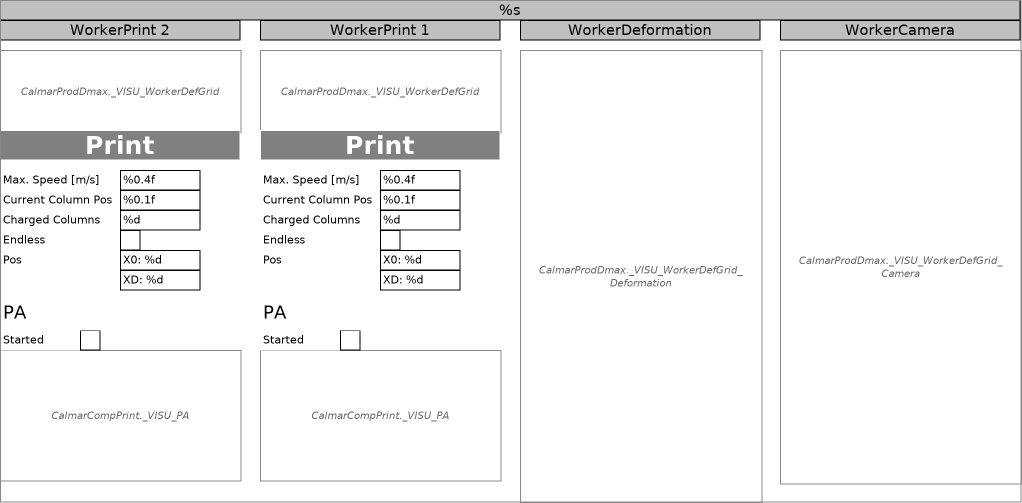
VISUALIZATION _VISU_Pm_Worker  // 1022x503
VAR_IN_OUT
	mInst : FB_PrintModule_WEU;
END_VAR
    Frame (0,50 242x404)
        shows _VISU_WorkerPrint_WEU(m_Inst := mInst.fbWorkerPrint[2])
    Frame (260,50 242x406)
        shows _VISU_WorkerPrint_WEU(m_Inst := mInst.fbWorkerPrint[1])
    Rectangle (0,20 240x20), "WorkerPrint 2"
    Rectangle (260,20 240x20), "WorkerPrint 1"
    Frame (780,50 242x434)
        shows CalmarProdDmax._VISU_WorkerDefGrid_Camera(m_Inst := mInst.fbWorkerCamera)
    Rectangle (780,20 240x20), "WorkerCamera"
    Rectangle (0,0 1020x20), "%s", text variable: mInst._pAdsPm^.aO_Name
    Rectangle (520,20 240x20), "WorkerDeformation"
    Frame (520,50 242x453)
        shows CalmarProdDmax._VISU_WorkerDefGrid_Deformation(m_Inst := mInst.fbWorkerDeformation)
END_VISUALIZATION

// ---- POUs/Projects/Machine/_VISU_MachineComm.TcVIS
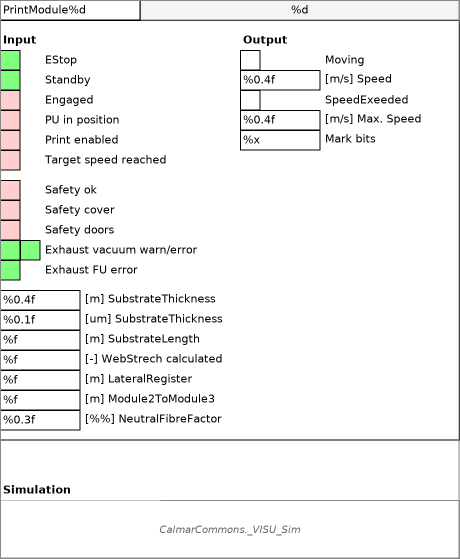
VISUALIZATION _VISU_MachineComm  // 460x559
VAR_IN_OUT
	mInst : FB_MachineComm;
END_VAR
    Rectangle (0,20 460x420)
    Frame (0,50 260x364)
        shows _VISU_MachineIn(ref := mInst.sModuleMachineState[mInst.nSelPm])
    Frame (240,50 214x110)
        shows _VISU_MachineOut(ref := mInst.sModuleMachineFeedback[mInst.nSelPm])
    Frame (0,500 460x59)
        shows CalmarCommons._VISU_Sim(mInst := mInst)
    Rectangle (240,30 160x20), "Output"
    Rectangle (0,30 160x20), "Input"
    Rectangle (0,480 160x20), "Simulation"
    Scrollbar (140,0 320x20), "%d", text variable: mInst.nSelPm
        p2245068023: iCPr_NB_PM
        p1057716461: mInst.nSelPm
    Rectangle (0,0 140x20), "PrintModule%d", text variable: PRG_PRINT.fbModuleMaster.nViewPmSel
END_VISUALIZATION

// ---- POUs/Projects/Machine/_VISU_MachineIn.TcVIS
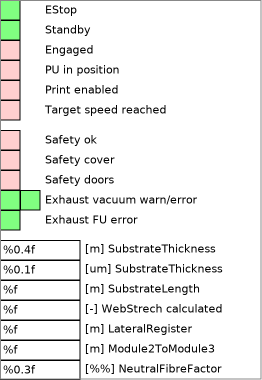
VISUALIZATION _VISU_MachineIn  // 262x380
VAR_IN_OUT
	ref : ST_ModuleMachineInterface_IN;
END_VAR
    Rectangle (0,320 80x20), "%f", text variable: ref.fLateralRegister
    Rectangle (82,320 180x18), "[m] LateralRegister"
    Rectangle (0,240 80x20), "%0.4f", text variable: ref.fSubstrateThickness
    Rectangle (82,240 180x18), "[m] SubstrateThickness"
    Rectangle (0,280 80x20), "%f", text variable: ref.fSubstrateLen
    Rectangle (82,280 180x18), "[m] SubstrateLength"
    Rectangle (0,300 80x20), "%f", text variable: ref.fWebStretchCalculated
    Rectangle (82,300 180x18), "[-] WebStrech calculated"
    Rectangle (0,340 80x20), "%f", text variable: ref.fModule2ToModule3
    Rectangle (82,340 180x18), "[m] Module2ToModule3"
    Rectangle (0,360 80x20), "%0.3f", text variable: ref.fNeutralFibreFactor
    Rectangle (82,360 180x18), "[%%] NeutralFibreFactor"
    Rectangle (42,20 180x20), "Standby"
    RoundedRectangle (0,0 20x20), colour toggle: ref.bEStop
    Rectangle (42,0 180x20), "EStop"
    RoundedRectangle (0,20 20x20), colour toggle: ref.bSleep
    RoundedRectangle (0,150 20x20), colour toggle: ref.bSafetyCoverOk
    Rectangle (42,150 180x20), "Safety cover"
    RoundedRectangle (0,170 20x20), colour toggle: ref.bServiceDoorsOk
    Rectangle (42,170 180x20), "Safety doors"
    RoundedRectangle (0,190 20x20), colour toggle: ref.bExhaustVacuumWarning
    Rectangle (42,190 180x20), "Exhaust vacuum warn/error"
    Rectangle (42,210 180x20), "Exhaust FU error"
    Rectangle (42,130 180x20), "Safety ok"
    RoundedRectangle (0,130 20x20), colour toggle: ref.bSafetyOk
    RoundedRectangle (20,190 20x20), colour toggle: ref.bExhaustVacuumError
    RoundedRectangle (0,210 20x20), colour toggle: ref.bExhaustFUError
    Rectangle (42,60 180x20), "PU in position"
    RoundedRectangle (0,60 20x20), colour toggle: ref.bUnitInPrintPosition
    Rectangle (42,40 180x20), "Engaged"
    RoundedRectangle (0,40 20x20), colour toggle: ref.bEngaged
    Rectangle (42,80 180x20), "Print enabled"
    RoundedRectangle (0,80 20x20), colour toggle: ref.bPrintEnabled
    Rectangle (42,100 180x20), "Target speed reached"
    RoundedRectangle (0,100 20x20), colour toggle: ref.bTargetSpeedReached
    Rectangle (0,260 80x20), "%0.1f", text variable: ref.fSubstrateThickness * 1_000_000
    Rectangle (82,260 180x18), "[um] SubstrateThickness"
END_VISUALIZATION

// ---- POUs/Projects/Machine/_VISU_MachineOut.TcVIS
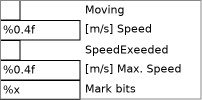
VISUALIZATION _VISU_MachineOut  // 202x100
VAR_IN_OUT
	ref : ST_ModuleMachineInterface_OUT;
END_VAR
    Rectangle (0,20 80x20), "%0.4f", text variable: ref.fSpeed
    Rectangle (82,20 120x18), "[m/s] Speed"
    Rectangle (0,60 80x20), "%0.4f", text variable: ref.fMaxSpeed
    Rectangle (82,60 120x18), "[m/s] Max. Speed"
    Rectangle (82,0 120x20), "Moving"
    RoundedRectangle (0,40 20x20), colour toggle: ref.bSpeedExeeded
    Rectangle (82,40 120x20), "SpeedExeeded"
    RoundedRectangle (0,0 20x20), colour toggle: ref.bMoving
    Rectangle (0,80 80x20), "%x", text variable: ref.nPrintMarkPosBits
    Rectangle (82,80 120x18), "Mark bits"
END_VISUALIZATION

// ---- POUs/Projects/Print/_Test/_VISU_PrgPrint_test.TcVIS
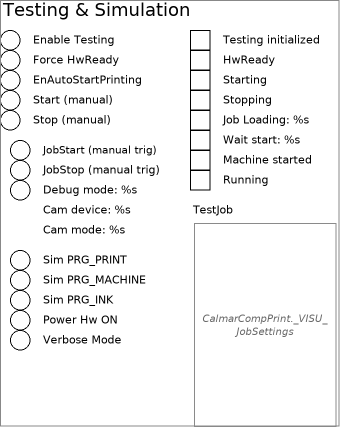
VISUALIZATION _VISU_PrgPrint_test  // 340x427
VAR_IN_OUT
	mInst : FB_PrgPrint_test;
END_VAR
    Ellipse (0,30 20x20)
        toggle mInst._bEnTesting
    Rectangle (30,30 120x20), "Enable Testing"
    Ellipse (0,70 20x20)
        toggle mInst._bEnAutoStartPrinting
    Rectangle (30,70 120x20), "EnAutoStartPrinting"
    Ellipse (10,180 20x20)
        toggle mInst._bEnVerboseMode
    Rectangle (40,180 120x20), "Debug mode: %s", text variable: mInst._eLogLevel
    Ellipse (10,270 20x20)
        toggle mInst._bSimPrgMachine
    Rectangle (40,270 120x20), "Sim PRG_MACHINE"
    Ellipse (10,290 20x20)
        toggle mInst._bSimPrgInk
    Rectangle (40,290 120x20), "Sim PRG_INK"
    Ellipse (10,250 20x20)
        toggle mInst._bSimPrgPrint
    Rectangle (40,250 120x20), "Sim PRG_PRINT"
    RoundedRectangle (190,30 20x20), colour toggle: mInst.bInitialized
    Rectangle (220,30 120x20), "Testing initialized"
    RoundedRectangle (190,50 20x20), tooltip "All enabled CBs are in OP", colour toggle: mInst.bHwReady
    Rectangle (220,50 120x20), "HwReady"
    RoundedRectangle (190,70 20x20), colour toggle: mInst.bStarting
    Rectangle (220,70 120x20), "Starting"
    RoundedRectangle (190,90 20x20), colour toggle: mInst.bStopping
    Rectangle (220,90 120x20), "Stopping"
    RoundedRectangle (190,170 20x20), colour toggle: mInst.bRunning
    Rectangle (220,170 120x20), "Running"
    Rectangle (220,110 120x20), "Job Loading: %s", tooltip "Timeout after: %s", text variable: mInst.LoadTestJob.tExecute.ET
        p4168582468: mInst.LoadTestJob.tExecute.PT
    RoundedRectangle (190,110 20x20), colour toggle: mInst.LoadTestJob.bbusy
    Rectangle (220,130 120x20), "Wait start: %s", text variable: mInst.TestStartSequence.tWaitJobStart.ET
    RoundedRectangle (190,130 20x20), colour toggle: mInst.TestStartSequence.tWaitJobStart.IN
    Rectangle (40,200 120x20), "Cam device: %s", text variable: mInst.eCameraDevice
        OnMouseClick: write the text variable via Default
    Rectangle (40,220 120x20), "Cam mode: %s", text variable: mInst.eCameraMode
        OnMouseClick: write the text variable via Default
    Ellipse (0,90 20x20)
        toggle mInst.bStart
    Rectangle (30,90 120x20), "Start (manual)"
    Ellipse (0,110 20x20)
        toggle mInst.bStop
    Rectangle (30,110 120x20), "Stop (manual)"
    Rectangle (0,0 200x20), "Testing & Simulation"
    Ellipse (10,140 20x20)
        tap mInst._pAdsPu^.sI_Start.bI_Command
        toggle mInst.bStart
    Rectangle (40,140 120x20), "JobStart (manual trig)"
    Ellipse (10,160 20x20)
        tap mInst._pAdsPu^.sI_Stop.bI_Command
        toggle mInst.bStop
    Rectangle (40,160 120x20), "JobStop (manual trig)"
    Frame (194,223 142x204)
        shows CalmarCompPrint._VISU_JobSettings(mInst := mInst.sJobConfig)
    RoundedRectangle (190,150 20x20), colour toggle: mInst.bRunMachine
    Rectangle (220,150 120x20), "Machine started"
    Rectangle (190,200 120x20), "TestJob"
    Ellipse (0,50 20x20)
        toggle mInst._bForceHwReady
    Rectangle (30,50 120x20), "Force HwReady"
    Ellipse (10,310 20x20)
        toggle mInst.bO_Power24V_ON
    Rectangle (40,310 120x20), "Power Hw ON"
    Ellipse (10,330 20x20)
        toggle mInst._bEnVerboseMode
    Rectangle (40,330 120x20), "Verbose Mode"
END_VISUALIZATION

// ---- VISUs/Projects/InkSystem/VISU_ADS_INKSTORAGE_TANK_DVT.TcVIS
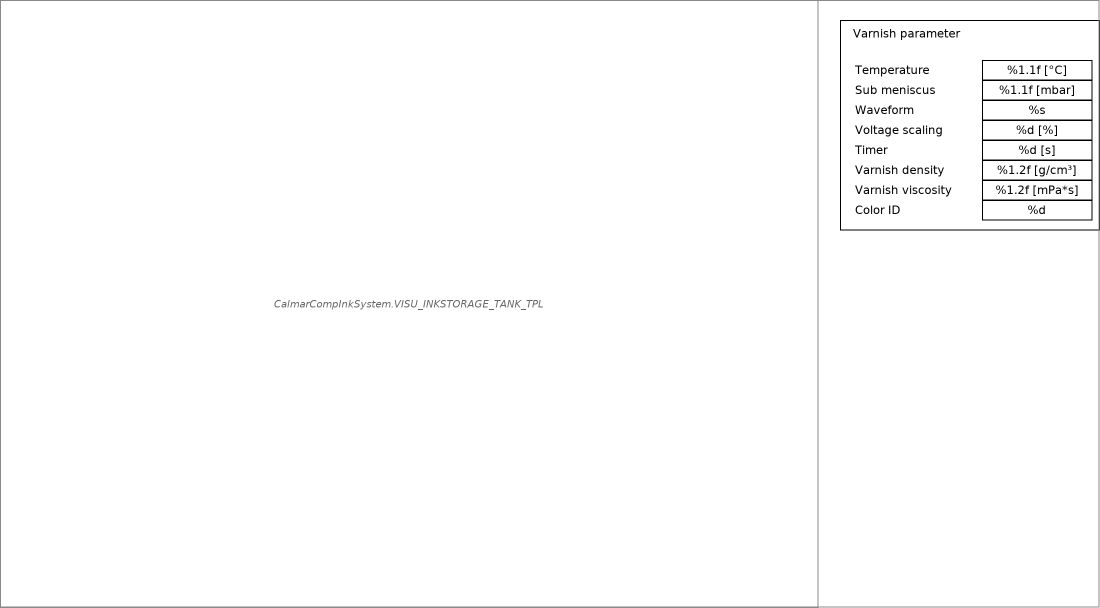
VISUALIZATION VISU_ADS_INKSTORAGE_TANK_DVT  // 1100x608
    Frame (0,0 818x608)
        shows CalmarCompInkSystem.VISU_INKSTORAGE_TANK_TPL(m_Idx_Max := CONFIGURATION.iCIk_NB_INKSTORAGE_TANK, m_ModId_StAdsStorageTank := PRG_INK.sAdsIkInkStorageTank[PRG_INK.iL_Sel_InkStorTank], m_Idx := PRG_INK.iL_Sel_InkStorTank, m_EnableBalanceLink := PRG_INK.bI_EnableBalanceLink, m_RefreshRate := PRG_INK.iI_RefreshRate, m_BalanceOffset := PRG_INK.fL_BalanceOffset[PRG_INK.iL_Sel_InkStorTank], m_CorrectionValue := PRG_INK.fI_CorrectionValue, m_MixerFeedbackExist := PRG_INK.bL_MixerFeedbackExist, m_MixerPulseIndicator := PRG_INK.bL_MixerPulseIndicator[PRG_INK.iL_Sel_InkStorTank], m_AckMixerPulseError := PRG_INK.bL_AckMixerPulseError[PRG_INK.iL_Sel_InkStorTank], m_MixerOnTime := PRG_INK.fL_MixerOnTime, m_MixerWaitTime := PRG_INK.fL_MixerWaitTime)
    Rectangle (840,20 260x210)
    Rectangle (982,60 110x20), "%1.1f [°C]", text variable: PRG_INK.sAdsIkInkStorageTank[PRG_INK.iL_Sel_InkStorTank].sI_InkParameter.sTemperature.fI_Val
        OnMouseDown: write the text variable via Edit, min PRG_INK.sAdsIkInkStorageTank[PRG_INK.iL_Sel_InkStorTank].sI_MaintenanceTimeout.lC_Min, max PRG_INK.sAdsIkInkStorageTank[PRG_INK.iL_Sel_InkStorTank].sI_MaintenanceTimeout.lC_Max
    Rectangle (852,60 130x20), "Temperature"
    Rectangle (850,25 191x17), "Varnish parameter"
    Rectangle (982,80 110x20), "%1.1f [mbar]", text variable: PRG_INK.sAdsIkInkStorageTank[PRG_INK.iL_Sel_InkStorTank].sI_InkParameter.sMeniscus.fI_Val
        OnMouseDown: write the text variable via Edit, min PRG_INK.sAdsIkInkStorageTank[PRG_INK.iL_Sel_InkStorTank].sI_InkParameter.sMeniscus.fC_Min, max PRG_INK.sAdsIkInkStorageTank[PRG_INK.iL_Sel_InkStorTank].sI_InkParameter.sMeniscus.fC_Max
    Rectangle (852,80 130x20), "Sub meniscus"
    Rectangle (982,100 110x20), "%s", text variable: PRG_INK.sAdsIkInkStorageTank[PRG_INK.iL_Sel_InkStorTank].sI_InkParameter.aWaveform
        OnMouseDown: write the text variable via Edit, min PRG_INK.sAdsIkInkStorageTank[PRG_INK.iL_Sel_InkStorTank].sI_MaintenanceTimeout.lC_Min, max PRG_INK.sAdsIkInkStorageTank[PRG_INK.iL_Sel_InkStorTank].sI_MaintenanceTimeout.lC_Max
    Rectangle (852,100 130x20), "Waveform"
    Rectangle (982,120 110x20), "%d [%]", text variable: PRG_INK.sAdsIkInkStorageTank[PRG_INK.iL_Sel_InkStorTank].sI_InkParameter.iVoltage
        OnMouseDown: write the text variable via Edit, min PRG_INK.sAdsIkInkStorageTank[PRG_INK.iL_Sel_InkStorTank].sI_MaintenanceTimeout.lC_Min, max PRG_INK.sAdsIkInkStorageTank[PRG_INK.iL_Sel_InkStorTank].sI_MaintenanceTimeout.lC_Max
    Rectangle (852,120 130x20), "Voltage scaling"
    Rectangle (982,140 110x20), "%d [s]", text variable: PRG_INK.sAdsIkInkStorageTank[PRG_INK.iL_Sel_InkStorTank].sI_InkParameter.iTimer
        OnMouseDown: write the text variable via Edit, min PRG_INK.sAdsIkInkStorageTank[PRG_INK.iL_Sel_InkStorTank].sI_MaintenanceTimeout.lC_Min, max PRG_INK.sAdsIkInkStorageTank[PRG_INK.iL_Sel_InkStorTank].sI_MaintenanceTimeout.lC_Max
    Rectangle (852,140 130x20), "Timer"
    Rectangle (982,160 110x20), "%1.2f [g/cm³]", text variable: PRG_INK.sAdsIkInkStorageTank[PRG_INK.iL_Sel_InkStorTank].sI_InkParameter.sDensity.fI_Val
        OnMouseDown: write the text variable via Edit, min PRG_INK.sAdsIkInkStorageTank[PRG_INK.iL_Sel_InkStorTank].sI_MaintenanceTimeout.lC_Min, max PRG_INK.sAdsIkInkStorageTank[PRG_INK.iL_Sel_InkStorTank].sI_MaintenanceTimeout.lC_Max
    Rectangle (852,160 130x20), "Varnish density"
    Rectangle (982,180 110x20), "%1.2f [mPa*s]", text variable: PRG_INK.sAdsIkInkStorageTank[PRG_INK.iL_Sel_InkStorTank].sI_InkParameter.sViscosity.fI_Val
        OnMouseDown: write the text variable via Edit, min PRG_INK.sAdsIkInkStorageTank[PRG_INK.iL_Sel_InkStorTank].sI_MaintenanceTimeout.lC_Min, max PRG_INK.sAdsIkInkStorageTank[PRG_INK.iL_Sel_InkStorTank].sI_MaintenanceTimeout.lC_Max
    Rectangle (852,180 130x20), "Varnish viscosity"
    Rectangle (982,200 110x20), "%d", text variable: PRG_INK.sAdsIkInkStorageTank[PRG_INK.iL_Sel_InkStorTank].sI_InkParameter.iColorId
        OnMouseDown: write the text variable via Edit, min PRG_INK.sAdsIkInkStorageTank[PRG_INK.iL_Sel_InkStorTank].sI_MaintenanceTimeout.lC_Min, max PRG_INK.sAdsIkInkStorageTank[PRG_INK.iL_Sel_InkStorTank].sI_MaintenanceTimeout.lC_Max
    Rectangle (852,200 130x20), "Color ID"
END_VISUALIZATION

// ---- VISUs/Projects/InkSystem/VISU_BALANCE.TcVIS
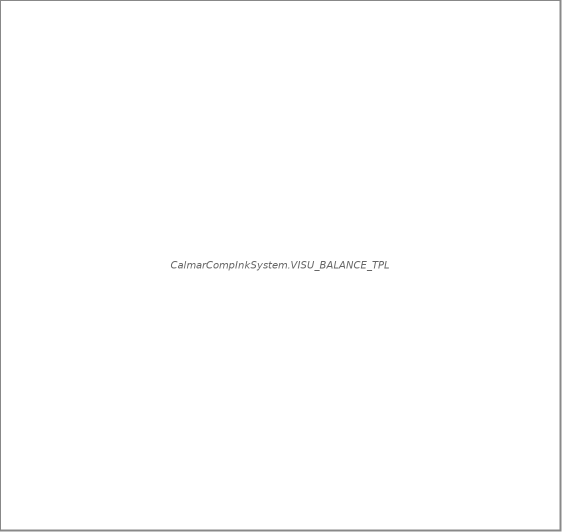
VISUALIZATION VISU_BALANCE  // 562x532
    Frame (0,0 560x530)
        shows CalmarCompInkSystem.VISU_BALANCE_TPL(m_Idx_Max := CONFIGURATION.iCIk_NB_INKBALANCE, m_ModId_StAdsStorageTank := PRG_INK.sAdsIkInkStorageTank[PRG_INK.iL_SelectedBalance], m_ModId_FbBalanceMonitor := PRG_INK.FB_Balance[PRG_INK.iL_SelectedBalance], m_Idx := PRG_INK.iL_SelectedBalance)
END_VISUALIZATION

// ---- VISUs/Projects/InkSystem/VISU_BARCODE.TcVIS
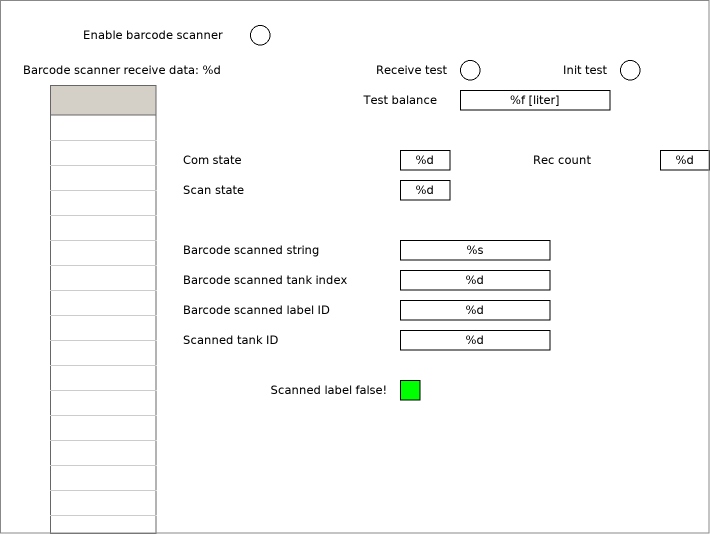
VISUALIZATION VISU_BARCODE  // 710x534
    Table (50,85 106x449), data array: PRG_INK.cI_Barcode_RxBuff
        p2232123230: PRG_INK.cI_Barcode_RxBuff[INDEX]
        p511219082: PRG_PRINT.sL_SensorResults[INDEX].yMark
        p1755163831: PRG_PRINT.sL_SensorResults[INDEX].phiMark
        p4092479075: PRG_PRINT.sL_SensorResults[INDEX].xCam
        p2237128397: PRG_PRINT.sL_SensorResults[INDEX].yCam
        p505689113: PRG_PRINT.sL_SensorResults[INDEX].phiCam
        p1757482276: PRG_PRINT.sL_SensorResults[INDEX].dx
        p4088588272: PRG_PRINT.sL_SensorResults[INDEX].dy
        p2243050616: PRG_PRINT.sL_SensorResults[INDEX].dphi
    Rectangle (20,60 240x20), "Barcode scanner receive data: %d", text variable: PRG_INK.iI_Barcode_RecDataLength
    Rectangle (400,240 150x20), "%s", text variable: PRG_INK.fb_BarcodeStoragetank.aL_ReceivedData
    Rectangle (180,240 200x20), "Barcode scanned string"
    Rectangle (400,270 150x20), "%d", text variable: PRG_INK.fb_BarcodeStoragetank.iL_ScannedStorageIndex
    Rectangle (180,270 200x20), "Barcode scanned tank index"
    Rectangle (400,300 150x20), "%d", text variable: PRG_INK.fb_BarcodeStoragetank.lL_ScannedLabel
    Rectangle (180,300 200x20), "Barcode scanned label ID"
    Rectangle (400,330 150x20), "%d", text variable: PRG_INK.sAdsIkInkStorageTank[PRG_INK.fb_BarcodeStoragetank.iL_ScannedStorageIndex].sI_InkParameter.iScannerId
        OnMouseClick: write the text variable via Default
    Rectangle (180,330 200x20), "Scanned tank ID"
    Rectangle (219,380 171x20), "Scanned label false!"
    RoundedRectangle (400,380 20x20), colour toggle: PRG_INK.fb_BarcodeStoragetank.bO_LabelScanFalse[PRG_INK.fb_BarcodeStoragetank.iL_ScannedStorageIndex]
    Rectangle (80,25 160x20), "Enable barcode scanner"
    Ellipse (250,25 20x20), colour toggle: PRG_INK.bI_EnableBarcodeScanner
        toggle PRG_INK.bI_EnableBarcodeScanner
    Rectangle (355,60 95x20), "Receive test"
    Ellipse (460,60 20x20), colour toggle: PRG_INK.bI_Barcode_DataRec
        tap PRG_INK.bI_Barcode_DataRec
    Rectangle (400,180 50x20), "%d", text variable: PRG_INK.fb_BarcodeStoragetank.iL_ScanState
        OnMouseClick: write the text variable via Default
    Rectangle (180,180 200x20), "Scan state"
    Rectangle (515,60 95x20), "Init test"
    Ellipse (620,60 20x20), colour toggle: PRG_INK.bI_Barcode_AckInit
        tap PRG_INK.bI_Barcode_AckInit
    Rectangle (400,150 50x20), "%d", text variable: PRG_INK.fb_BarcodeStoragetank.iL_COMstate
        OnMouseClick: write the text variable via Default
    Rectangle (180,150 200x20), "Com state"
    Rectangle (460,90 150x20), "%f [liter]", text variable: PRG_INK.FB_BalanceLink.fO_Readings[PRG_INK.fb_BarcodeStoragetank.iL_ScannedStorageIndex]
        OnMouseClick: write the text variable via Default
    Rectangle (329,90 111x20), "Test balance"
    Rectangle (660,150 50x20), "%d", text variable: PRG_INK.fb_BarcodeStoragetank.iL_ReceiveCount
    Rectangle (530,150 102x20), "Rec count"
END_VISUALIZATION

// ---- VISUs/Projects/InkSystem/VISU_COMM_BALANCE.TcVIS
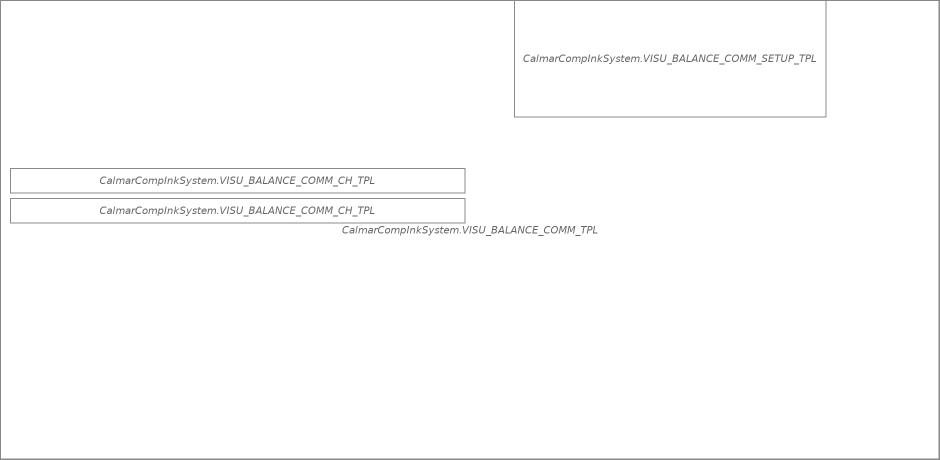
VISUALIZATION VISU_COMM_BALANCE  // 940x460
    Frame (0,0 940x460)
        shows CalmarCompInkSystem.VISU_BALANCE_COMM_TPL(m_ModId_FbBalanceComm := PRG_INK.FB_BalanceLink)
    Frame (514,0 312x117)
        shows CalmarCompInkSystem.VISU_BALANCE_COMM_SETUP_TPL(m_ModId_FbBalanceComm := PRG_INK.FB_BalanceLink)
    Frame (10,168 455x25)
        shows CalmarCompInkSystem.VISU_BALANCE_COMM_CH_TPL(m_Idx := 1, m_ModId_StAdsStorageTank := PRG_INK.sAdsIkInkStorageTank[1], m_ModId_StInkDefinition := PRG_INK.sL_InkTable[1], m_ModId_FbBalanceComm := PRG_INK.FB_BalanceLink)
    Frame (10,198 455x25)
        shows CalmarCompInkSystem.VISU_BALANCE_COMM_CH_TPL(m_Idx := 2, m_ModId_StAdsStorageTank := PRG_INK.sAdsIkInkStorageTank[2], m_ModId_StInkDefinition := PRG_INK.sL_InkTable[2], m_ModId_FbBalanceComm := PRG_INK.FB_BalanceLink)
END_VISUALIZATION

// ---- VISUs/Projects/InkSystem/VISU_HEADERTANK.TcVIS
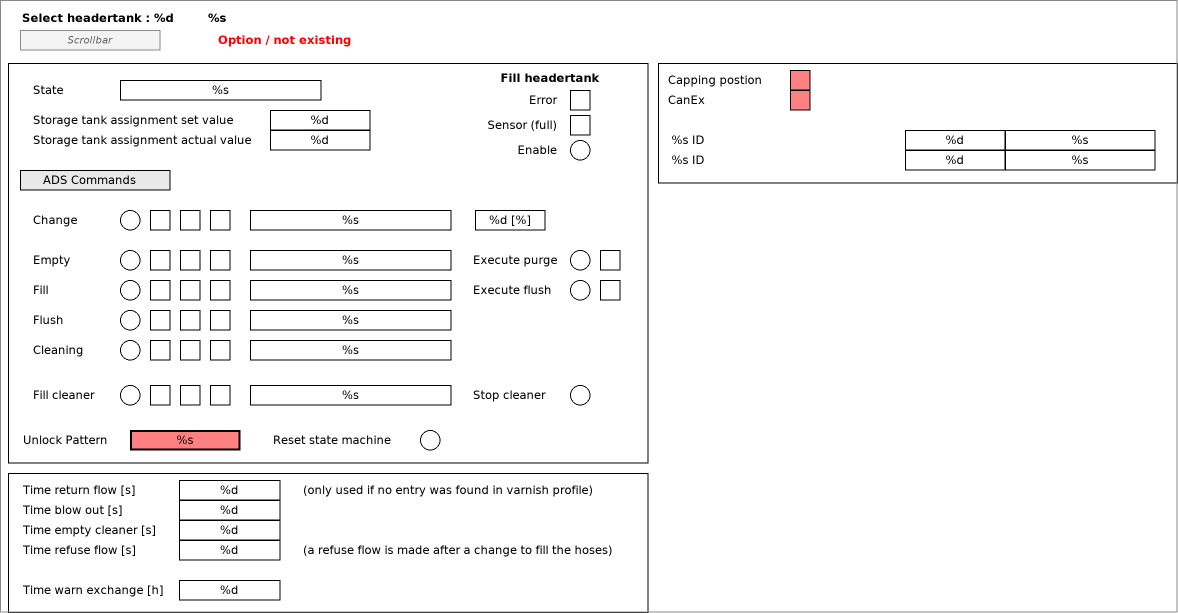
VISUALIZATION VISU_HEADERTANK  // 1178x613
    Rectangle (658,63 520x120)
    Rectangle (8,473 640x140)
    Rectangle (8,63 640x400)
    Rectangle (30,310 80x20), "Flush"
    Ellipse (120,310 20x20), colour toggle: PRG_INK.sAdsIkHeaderTank[PRG_INK.iL_Sel_HeaderTank].sI_CommandFlush.bI_Command, input disabled if: NOT PRG_INK.sAdsIkHeaderTank[PRG_INK.iL_Sel_HeaderTank].sI_CommandFlush.bO_CommandCanEx
        tap PRG_INK.sAdsIkHeaderTank[PRG_INK.iL_Sel_HeaderTank].sI_CommandFlush.bI_Command
    Rectangle (20,170 150x20)
    Rectangle (40,170 130x20), "ADS Commands"
    RoundedRectangle (150,310 20x20), tooltip "CanEx", colour toggle: PRG_INK.sAdsIkHeaderTank[PRG_INK.iL_Sel_HeaderTank].sI_CommandFlush.bO_CommandCanEx
    RoundedRectangle (210,310 20x20), tooltip "Exec", colour toggle: PRG_INK.sAdsIkHeaderTank[PRG_INK.iL_Sel_HeaderTank].sI_CommandFlush.bO_CommandExec
    RoundedRectangle (180,310 20x20), tooltip "CanStop", colour toggle: PRG_INK.sAdsIkHeaderTank[PRG_INK.iL_Sel_HeaderTank].sI_CommandFlush.bO_CommandCanStop
    Scrollbar (20,30 140x20), tooltip "y-shift"
        p2245068023: CONFIGURATION.iCIk_NB_HEADERTANK
        p1057716461: PRG_INK.iL_Sel_HeaderTank
    Rectangle (15,8 180x20), "Select headertank : %d", text variable: PRG_INK.iL_Sel_HeaderTank
    Rectangle (30,340 80x20), "Cleaning"
    Ellipse (120,340 20x20), colour toggle: PRG_INK.sAdsIkHeaderTank[PRG_INK.iL_Sel_HeaderTank].sI_CommandCleaning.bI_Command, input disabled if: NOT PRG_INK.sAdsIkHeaderTank[PRG_INK.iL_Sel_HeaderTank].sI_CommandCleaning.bO_CommandCanEx
        tap PRG_INK.sAdsIkHeaderTank[PRG_INK.iL_Sel_HeaderTank].sI_CommandCleaning.bI_Command
    RoundedRectangle (150,340 20x20), tooltip "CanEx", colour toggle: PRG_INK.sAdsIkHeaderTank[PRG_INK.iL_Sel_HeaderTank].sI_CommandCleaning.bO_CommandCanEx
    RoundedRectangle (210,340 20x20), tooltip "Exec", colour toggle: PRG_INK.sAdsIkHeaderTank[PRG_INK.iL_Sel_HeaderTank].sI_CommandCleaning.bO_CommandExec
    RoundedRectangle (180,340 20x20), tooltip "CanStop", colour toggle: PRG_INK.sAdsIkHeaderTank[PRG_INK.iL_Sel_HeaderTank].sI_CommandCleaning.bO_CommandCanStop
    Rectangle (30,280 80x20), "Fill"
    Ellipse (120,280 20x20), colour toggle: PRG_INK.sAdsIkHeaderTank[PRG_INK.iL_Sel_HeaderTank].sI_CommandFill.bI_Command, input disabled if: NOT PRG_INK.sAdsIkHeaderTank[PRG_INK.iL_Sel_HeaderTank].sI_CommandFill.bO_CommandCanEx
        tap PRG_INK.sAdsIkHeaderTank[PRG_INK.iL_Sel_HeaderTank].sI_CommandFill.bI_Command
    RoundedRectangle (150,280 20x20), tooltip "CanEx", colour toggle: PRG_INK.sAdsIkHeaderTank[PRG_INK.iL_Sel_HeaderTank].sI_CommandFill.bO_CommandCanEx
    RoundedRectangle (210,280 20x20), tooltip "Exec", colour toggle: PRG_INK.sAdsIkHeaderTank[PRG_INK.iL_Sel_HeaderTank].sI_CommandFill.bO_CommandExec
    RoundedRectangle (180,280 20x20), tooltip "CanStop", colour toggle: PRG_INK.sAdsIkHeaderTank[PRG_INK.iL_Sel_HeaderTank].sI_CommandFill.bO_CommandCanStop
    Rectangle (30,250 80x20), "Empty"
    Ellipse (120,250 20x20), colour toggle: PRG_INK.sAdsIkHeaderTank[PRG_INK.iL_Sel_HeaderTank].sI_CommandEmpty.bI_Command, input disabled if: NOT PRG_INK.sAdsIkHeaderTank[PRG_INK.iL_Sel_HeaderTank].sI_CommandEmpty.bO_CommandCanEx
        tap PRG_INK.sAdsIkHeaderTank[PRG_INK.iL_Sel_HeaderTank].sI_CommandEmpty.bI_Command
    RoundedRectangle (150,250 20x20), tooltip "CanEx", colour toggle: PRG_INK.sAdsIkHeaderTank[PRG_INK.iL_Sel_HeaderTank].sI_CommandEmpty.bO_CommandCanEx
    RoundedRectangle (210,250 20x20), tooltip "Exec", colour toggle: PRG_INK.sAdsIkHeaderTank[PRG_INK.iL_Sel_HeaderTank].sI_CommandEmpty.bO_CommandExec
    RoundedRectangle (180,250 20x20), tooltip "CanStop", colour toggle: PRG_INK.sAdsIkHeaderTank[PRG_INK.iL_Sel_HeaderTank].sI_CommandEmpty.bO_CommandCanStop
    Rectangle (250,250 201x20), "%s", text variable: PRG_INK.fb_Headertank[PRG_INK.iL_Sel_HeaderTank].aL_StateEmpty
    Rectangle (250,280 201x20), "%s", text variable: PRG_INK.fb_Headertank[PRG_INK.iL_Sel_HeaderTank].aL_StateFill
    Rectangle (250,310 201x20), "%s", text variable: PRG_INK.fb_Headertank[PRG_INK.iL_Sel_HeaderTank].aL_StateFlush
    Rectangle (250,340 201x20), "%s", text variable: PRG_INK.fb_Headertank[PRG_INK.iL_Sel_HeaderTank].aL_StateCleaning
    Rectangle (470,280 90x20), "Execute flush"
    Ellipse (570,280 20x20), colour toggle: PRG_INK.fb_Headertank[PRG_INK.iL_Sel_HeaderTank].bL_ExecuteFlushManu
        toggle PRG_INK.fb_Headertank[PRG_INK.iL_Sel_HeaderTank].bL_ExecuteFlushManu
    Rectangle (30,210 80x20), "Change"
    Ellipse (120,210 20x20), colour toggle: PRG_INK.sAdsIkHeaderTank[PRG_INK.iL_Sel_HeaderTank].sI_CommandChange.bI_Command, input disabled if: NOT PRG_INK.sAdsIkHeaderTank[PRG_INK.iL_Sel_HeaderTank].sI_CommandChange.bO_CommandCanEx
        tap PRG_INK.sAdsIkHeaderTank[PRG_INK.iL_Sel_HeaderTank].sI_CommandChange.bI_Command
    RoundedRectangle (150,210 20x20), tooltip "CanEx", colour toggle: PRG_INK.sAdsIkHeaderTank[PRG_INK.iL_Sel_HeaderTank].sI_CommandChange.bO_CommandCanEx
    RoundedRectangle (210,210 20x20), tooltip "Exec", colour toggle: PRG_INK.sAdsIkHeaderTank[PRG_INK.iL_Sel_HeaderTank].sI_CommandChange.bO_CommandExec
    RoundedRectangle (180,210 20x20), tooltip "CanStop", colour toggle: PRG_INK.sAdsIkHeaderTank[PRG_INK.iL_Sel_HeaderTank].sI_CommandChange.bO_CommandCanStop
    Rectangle (250,210 201x20), "%s", text variable: PRG_INK.fb_Headertank[PRG_INK.iL_Sel_HeaderTank].aL_StateChange
    Rectangle (270,110 100x20), "%d", text variable: PRG_INK.sAdsIkHeaderTank[PRG_INK.iL_Sel_HeaderTank].sI_StoragetankAssignment.lI_Val
        OnMouseDown: write the text variable via Default
    Rectangle (30,110 230x20), "Storage tank assignment set value"
    Rectangle (270,130 100x20), "%d", text variable: PRG_INK.sAdsIkHeaderTank[PRG_INK.iL_Sel_HeaderTank].sO_ActStoragetankAssignment.lI_Val
        OnMouseDown: write the text variable via Edit
    Rectangle (30,130 230x20), "Storage tank assignment actual value"
    RoundedRectangle (600,280 20x20), colour toggle: PRG_INK.fb_Headertank[PRG_INK.iL_Sel_HeaderTank].bL_ExecuteFlush
    Rectangle (120,80 201x20), "%s", text variable: PRG_INK.fb_Headertank[PRG_INK.iL_Sel_HeaderTank].eL_StateHeadertank
    Rectangle (179,480 101x20), "%d", text variable: PRG_INK.lL_TimeReturnFlow
        OnMouseDown: write the text variable via Edit
    Rectangle (20,480 147x20), "Time return flow [s]"
    Rectangle (179,500 101x20), "%d", text variable: PRG_INK.lL_TimeBlowOut
        OnMouseDown: write the text variable via Edit
    Rectangle (20,500 147x20), "Time blow out [s]"
    Rectangle (179,520 101x20), "%d", text variable: PRG_INK.lL_TimeEmptyCleaner
        OnMouseDown: write the text variable via Edit
    Rectangle (20,520 147x20), "Time empty cleaner [s]"
    Rectangle (179,580 101x20), "%d", text variable: PRG_INK.lL_TimeWarnExchange
        OnMouseDown: write the text variable via Edit
    Rectangle (20,580 147x20), "Time warn exchange [h]"
    Rectangle (470,90 90x20), "Error"
    RoundedRectangle (570,90 20x20), colour toggle: PRG_INK.sAdsIkHeaderTank[PRG_INK.iL_Sel_HeaderTank].sI_AckFillInk.bO_CommandCanEx
    Rectangle (30,80 80x20), "State"
    Ellipse (570,140 20x20), colour toggle: PRG_INK.sAdsIkHeaderTank[PRG_INK.iL_Sel_HeaderTank].bI_EnableFillInk
        toggle PRG_INK.sAdsIkHeaderTank[PRG_INK.iL_Sel_HeaderTank].bI_EnableFillInk
    Rectangle (470,140 90x20), "Enable"
    Rectangle (470,115 90x20), "Sensor (full)"
    RoundedRectangle (570,115 20x20), colour toggle: (PRG_INK.sAdsIkHeaderTank[PRG_INK.iL_Sel_HeaderTank].cO_StatusFillInk.5) <> 0
    Rectangle (20,430 100x20), "Unlock Pattern"
    Rectangle (130,430 110x20), "%s", text variable: PRG_INK.fb_Headertank[PRG_INK.iL_Sel_HeaderTank].aI_SafePattern, colour toggle: PRG_INK.fb_Headertank[PRG_INK.iL_Sel_HeaderTank].bL_Unlock
        OnMouseDown: write the text variable via Edit
    Ellipse (420,430 20x20), colour toggle: PRG_INK.fb_Headertank[PRG_INK.iL_Sel_HeaderTank].fb_RTrigStateMachineReset.CLK, invisible if: NOT PRG_INK.fb_Headertank[PRG_INK.iL_Sel_HeaderTank].bL_Unlock
        tap PRG_INK.fb_Headertank[PRG_INK.iL_Sel_HeaderTank].fb_RTrigStateMachineReset.CLK
    Rectangle (270,430 140x20), "Reset state machine", invisible if: NOT PRG_INK.fb_Headertank[PRG_INK.iL_Sel_HeaderTank].bL_Unlock
    Rectangle (905,130 100x20), "%d", text variable: PRG_INK.sL_BLK_INKSTORAGE_TANK[1].iBlk_AdsId
        OnMouseDown: write the text variable via Edit
    Rectangle (665,130 230x20), "%s ID", text variable: PRG_INK.sAdsIkInkStorageTank[1].aO_Name
    RoundedRectangle (790,90 20x20), colour toggle: PRG_INK.bL_HeadertankCanEx
        toggle PRG_INK.sAdsIkHeaderTank[PRG_INK.iL_Sel_HeaderTank].bI_EnableFillInk
    Rectangle (665,90 110x20), "CanEx"
    Rectangle (300,480 300x20), "(only used if no entry was found in varnish profile)"
    Rectangle (475,210 70x20), "%d [%]", text variable: PRG_INK.fb_Headertank[PRG_INK.iL_Sel_HeaderTank].iL_PercentStateChange
        OnMouseDown: write the text variable via Edit
    Rectangle (495,68 110x20), "Fill headertank"
    Rectangle (30,385 80x20), "Fill cleaner"
    Ellipse (120,385 20x20), colour toggle: PRG_INK.sAdsIkHeaderTank[PRG_INK.iL_Sel_HeaderTank].sI_ActivateCleaner.bI_Command, input disabled if: NOT PRG_INK.sAdsIkHeaderTank[PRG_INK.iL_Sel_HeaderTank].sI_ActivateCleaner.bO_CommandCanEx
        tap PRG_INK.sAdsIkHeaderTank[PRG_INK.iL_Sel_HeaderTank].sI_ActivateCleaner.bI_Command
    RoundedRectangle (150,385 20x20), tooltip "CanEx", colour toggle: PRG_INK.sAdsIkHeaderTank[PRG_INK.iL_Sel_HeaderTank].sI_ActivateCleaner.bO_CommandCanEx
    RoundedRectangle (210,385 20x20), tooltip "Exec", colour toggle: PRG_INK.sAdsIkHeaderTank[PRG_INK.iL_Sel_HeaderTank].sI_ActivateCleaner.bO_CommandExec
    RoundedRectangle (180,385 20x20), tooltip "CanStop", colour toggle: PRG_INK.sAdsIkHeaderTank[PRG_INK.iL_Sel_HeaderTank].sI_ActivateCleaner.bO_CommandCanStop
    Rectangle (250,385 201x20), "%s", text variable: PRG_INK.fb_Headertank[PRG_INK.iL_Sel_HeaderTank].aL_StateCleaner
    RoundedRectangle (790,70 20x20), colour toggle: PRG_INK.iMachineInk[iCIk_MAP_HEADERTANK_HT_GROUP[PRG_INK.iL_Sel_HeaderTank]].pInCappingPos
        toggle PRG_INK.sAdsIkHeaderTank[PRG_INK.iL_Sel_HeaderTank].bI_EnableFillInk
    Rectangle (665,70 110x20), "Capping postion"
    Rectangle (215,30 150x20), "Option / not existing", invisible if: bCIk_HEADERTANK_EXIST[PRG_INK.iL_Sel_HeaderTank]
    Rectangle (470,385 90x20), "Stop cleaner"
    Ellipse (570,385 20x20), colour toggle: PRG_INK.bIDp_StopFillCleaner[PRG_INK.iL_Sel_HeaderTank]
        tap PRG_INK.bIDp_StopFillCleaner[PRG_INK.iL_Sel_HeaderTank]
    Rectangle (905,150 100x20), "%d", text variable: PRG_INK.sL_BLK_INKSTORAGE_TANK[2].iBlk_AdsId
        OnMouseDown: write the text variable via Edit
    Rectangle (665,150 230x20), "%s ID", text variable: PRG_INK.sAdsIkInkStorageTank[2].aO_Name
    Rectangle (205,8 180x20), "%s", text variable: PRG_INK.sC_Config_I.aC_HEADERTANKGROUP_NAME_DETAIL[iCIk_MAP_HEADERTANK_HT_GROUP[PRG_INK.iL_Sel_HeaderTank]]
    Rectangle (1005,130 150x20), "%s", text variable: PRG_INK.sAdsIkInkStorageTank[1].sI_InkParameter.aColorName
        OnMouseDown: write the text variable via Edit
    Rectangle (1005,150 150x20), "%s", text variable: PRG_INK.sAdsIkInkStorageTank[2].sI_InkParameter.aColorName
        OnMouseDown: write the text variable via Edit
    Rectangle (179,540 101x20), "%d", text variable: PRG_INK.lL_TimeRefuseFlow
        OnMouseDown: write the text variable via Edit
    Rectangle (20,540 147x20), "Time refuse flow [s]"
    Rectangle (300,540 344x20), "(a refuse flow is made after a change to fill the hoses)"
    Rectangle (470,250 96x20), "Execute purge"
    Ellipse (570,250 20x20), colour toggle: PRG_INK.fb_Headertank[PRG_INK.iL_Sel_HeaderTank].bI_ExecutePurgeManu
        toggle PRG_INK.fb_Headertank[PRG_INK.iL_Sel_HeaderTank].bI_ExecutePurgeManu
    RoundedRectangle (600,250 20x20), colour toggle: PRG_INK.fb_Headertank[PRG_INK.iL_Sel_HeaderTank].bL_SkipPurge
END_VISUALIZATION

// ---- VISUs/Projects/InkSystem/VISU_HT_FLUSHING_DEVICE.TcVIS
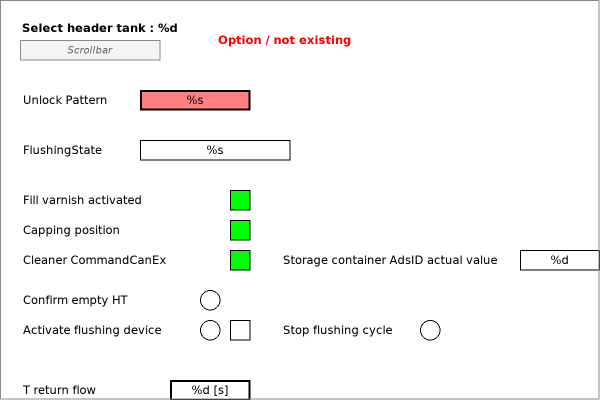
VISUALIZATION VISU_HT_FLUSHING_DEVICE  // 600x400
    Rectangle (20,190 160x20), "Fill varnish activated", invisible if: NOT PRG_INK.bL_FlushingUnlock
    Scrollbar (20,40 140x20), input disabled if: PRG_INK.bL_FlushingActive
        p2245068023: CONFIGURATION.iCIk_NB_HEADERTANK
        p1057716461: PRG_INK.iL_SelHeaderTankFlushing
    Rectangle (15,18 180x20), "Select header tank : %d", text variable: PRG_INK.iL_SelHeaderTankFlushing
    Rectangle (215,30 150x20), "Option / not existing", invisible if: bCIk_HEADERTANK_EXIST[PRG_INK.iL_SelHeaderTankFlushing]
    Rectangle (20,90 100x20), "Unlock Pattern"
    Rectangle (20,290 160x20), "Confirm empty HT", invisible if: NOT PRG_INK.bL_FlushingUnlock
    Rectangle (20,320 160x20), "Activate flushing device", invisible if: NOT PRG_INK.bL_FlushingUnlock
    Rectangle (20,380 110x20), "T return flow", invisible if: NOT PRG_INK.bL_FlushingUnlock
    Ellipse (200,320 20x20), colour toggle: PRG_INK.bL_FlushingActivate, invisible if: NOT PRG_INK.bL_FlushingUnlock
        toggle PRG_INK.bL_FlushingActivate
    RoundedRectangle (230,320 20x20), colour toggle: PRG_INK.bL_FlushingActive, invisible if: NOT PRG_INK.bL_FlushingUnlock
    Ellipse (200,290 20x20), colour toggle: PRG_INK.bL_FlushingHtEmpty, invisible if: NOT PRG_INK.bL_FlushingUnlock, input disabled if: NOT PRG_INK.bIKn_TankInkLevelReached[PRG_INK.iL_SelHeaderTankFlushing] OR PRG_INK.bL_FlushingActive
        toggle PRG_INK.bL_FlushingHtEmpty
    RoundedRectangle (230,190 20x20), colour toggle: PRG_INK.sAdsIkHeaderTank[PRG_INK.iL_SelHeaderTankFlushing].bI_EnableFillInk, invisible if: NOT PRG_INK.bL_FlushingUnlock
    Rectangle (170,380 80x20), "%d [s]", text variable: PRG_INK.lL_TimeFlushingReturnFlow, invisible if: NOT PRG_INK.bL_FlushingUnlock
        OnMouseDown: write the text variable via Edit
    Rectangle (140,90 110x20), "%s", text variable: PRG_INK.aI_FlushingSafePattern, colour toggle: PRG_INK.bL_FlushingUnlock
        OnMouseDown: write the text variable via Edit
    Rectangle (20,140 110x20), "FlushingState"
    Rectangle (140,140 150x20), "%s", text variable: PRG_INK.aL_FlushingState
    Rectangle (20,220 160x20), "Capping position", invisible if: NOT PRG_INK.bL_FlushingUnlock
    RoundedRectangle (230,220 20x20), colour toggle: NOT PRG_INK.bL_InCappingPos, invisible if: NOT PRG_INK.bL_FlushingUnlock
    Rectangle (280,320 130x20), "Stop flushing cycle", invisible if: NOT PRG_INK.bL_FlushingUnlock
    Ellipse (420,320 20x20), colour toggle: PRG_INK.bL_FlushingStop, invisible if: NOT PRG_INK.bL_FlushingUnlock
        toggle PRG_INK.bL_FlushingStop
    Rectangle (520,250 80x20), "%d", text variable: PRG_INK.sAdsIkHeaderTank[PRG_INK.iL_SelHeaderTankFlushing].sO_ActStoragetankAssignment.lI_Val, invisible if: NOT PRG_INK.bL_FlushingUnlock
        OnMouseDown: write the text variable via Edit
    Rectangle (280,250 230x20), "Storage container AdsID actual value", invisible if: NOT PRG_INK.bL_FlushingUnlock
    Rectangle (20,250 160x20), "Cleaner CommandCanEx", invisible if: NOT PRG_INK.bL_FlushingUnlock
    RoundedRectangle (230,250 20x20), colour toggle: NOT PRG_INK.sAdsIkHeaderTank[PRG_INK.iL_SelHeaderTankFlushing].sI_ActivateCleaner.bO_CommandCanEx, invisible if: NOT PRG_INK.bL_FlushingUnlock
END_VISUALIZATION

// ---- VISUs/Projects/InkSystem/VISU_INK.TcVIS
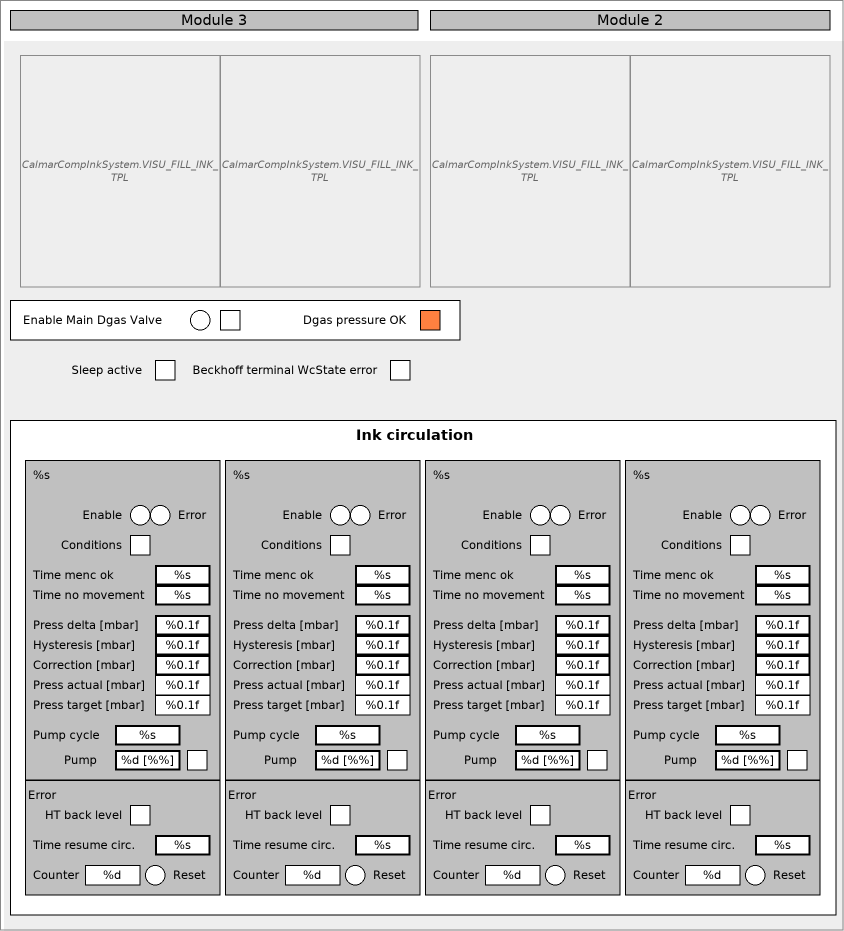
VISUALIZATION VISU_INK  // 844x931
    Rectangle (4,41 840x890)
    Rectangle (10,300 450x40)
    Ellipse (190,310 20x20), colour toggle: PRG_INK.bIDp_EnableMainDgasValve
        toggle PRG_INK.bIDp_EnableMainDgasValve
    Rectangle (20,310 160x20), "Enable Main Dgas Valve"
    RoundedRectangle (220,310 20x20), colour toggle: PRG_INK.bODp_EnableMainDgasValve
    Rectangle (300,310 110x20), "Dgas pressure OK"
    RoundedRectangle (420,310 20x20), colour toggle: PRG_INK.bODp_DgasPressOK
    RoundedRectangle (155,360 20x20), colour toggle: PRG_MACHINE.sO_SystemCmd.bSleep
    Rectangle (70,360 75x20), "Sleep active"
    RoundedRectangle (390,360 20x20), colour toggle: PRG_INK.bI_InkLevel1WcState
    Rectangle (190,360 190x20), "Beckhoff terminal WcState error"
    Frame (20,55 200x232)
        shows CalmarCompInkSystem.VISU_FILL_INK_TPL(m_InkDegasExisting := CONFIGURATION.bCIk_INK_DEGASSING_EXISTING, m_ModId_StAdsHeadertank := PRG_INK.sAdsIkHeaderTank[4], m_ModId_StAdsInkPump := PRG_INK.sAdsIkInkPump[4], m_ModId_FbInkSupply := PRG_INK.fb_FillInkVarnish[4], m_ModId_StInkDefinition := PRG_INK.sL_InkTable[4])
    Frame (220,55 200x232)
        shows CalmarCompInkSystem.VISU_FILL_INK_TPL(m_InkDegasExisting := CONFIGURATION.bCIk_INK_DEGASSING_EXISTING, m_ModId_StAdsHeadertank := PRG_INK.sAdsIkHeaderTank[3], m_ModId_StAdsInkPump := PRG_INK.sAdsIkInkPump[3], m_ModId_FbInkSupply := PRG_INK.fb_FillInkVarnish[3], m_ModId_StInkDefinition := PRG_INK.sL_InkTable[3])
    Frame (430,55 200x232)
        shows CalmarCompInkSystem.VISU_FILL_INK_TPL(m_InkDegasExisting := CONFIGURATION.bCIk_INK_DEGASSING_EXISTING, m_ModId_StAdsHeadertank := PRG_INK.sAdsIkHeaderTank[2], m_ModId_StAdsInkPump := PRG_INK.sAdsIkInkPump[2], m_ModId_FbInkSupply := PRG_INK.fb_FillInkVarnish[2], m_ModId_StInkDefinition := PRG_INK.sL_InkTable[2])
    Frame (630,55 200x232)
        shows CalmarCompInkSystem.VISU_FILL_INK_TPL(m_InkDegasExisting := CONFIGURATION.bCIk_INK_DEGASSING_EXISTING, m_ModId_StAdsHeadertank := PRG_INK.sAdsIkHeaderTank[1], m_ModId_StAdsInkPump := PRG_INK.sAdsIkInkPump[1], m_ModId_FbInkSupply := PRG_INK.fb_FillInkVarnish[1], m_ModId_StInkDefinition := PRG_INK.sL_InkTable[1])
    Rectangle (10,420 826x495)
    Rectangle (335,425 160x20), "Ink circulation"
    Frame (625,460 195x435)
        shows _VISU_InkCirculation(m_Inst_Fb := PRG_INK.fb_CirculationInk[1])
    Frame (425,460 195x435)
        shows _VISU_InkCirculation(m_Inst_Fb := PRG_INK.fb_CirculationInk[2])
    Frame (225,460 195x435)
        shows _VISU_InkCirculation(m_Inst_Fb := PRG_INK.fb_CirculationInk[3])
    Frame (25,460 195x435)
        shows _VISU_InkCirculation(m_Inst_Fb := PRG_INK.fb_CirculationInk[4])
    Rectangle (10,10 408x20), "Module 3"
    Rectangle (430,10 400x20), "Module 2"
END_VISUALIZATION

// ---- VISUs/Projects/InkSystem/VISU_PURGE.TcVIS
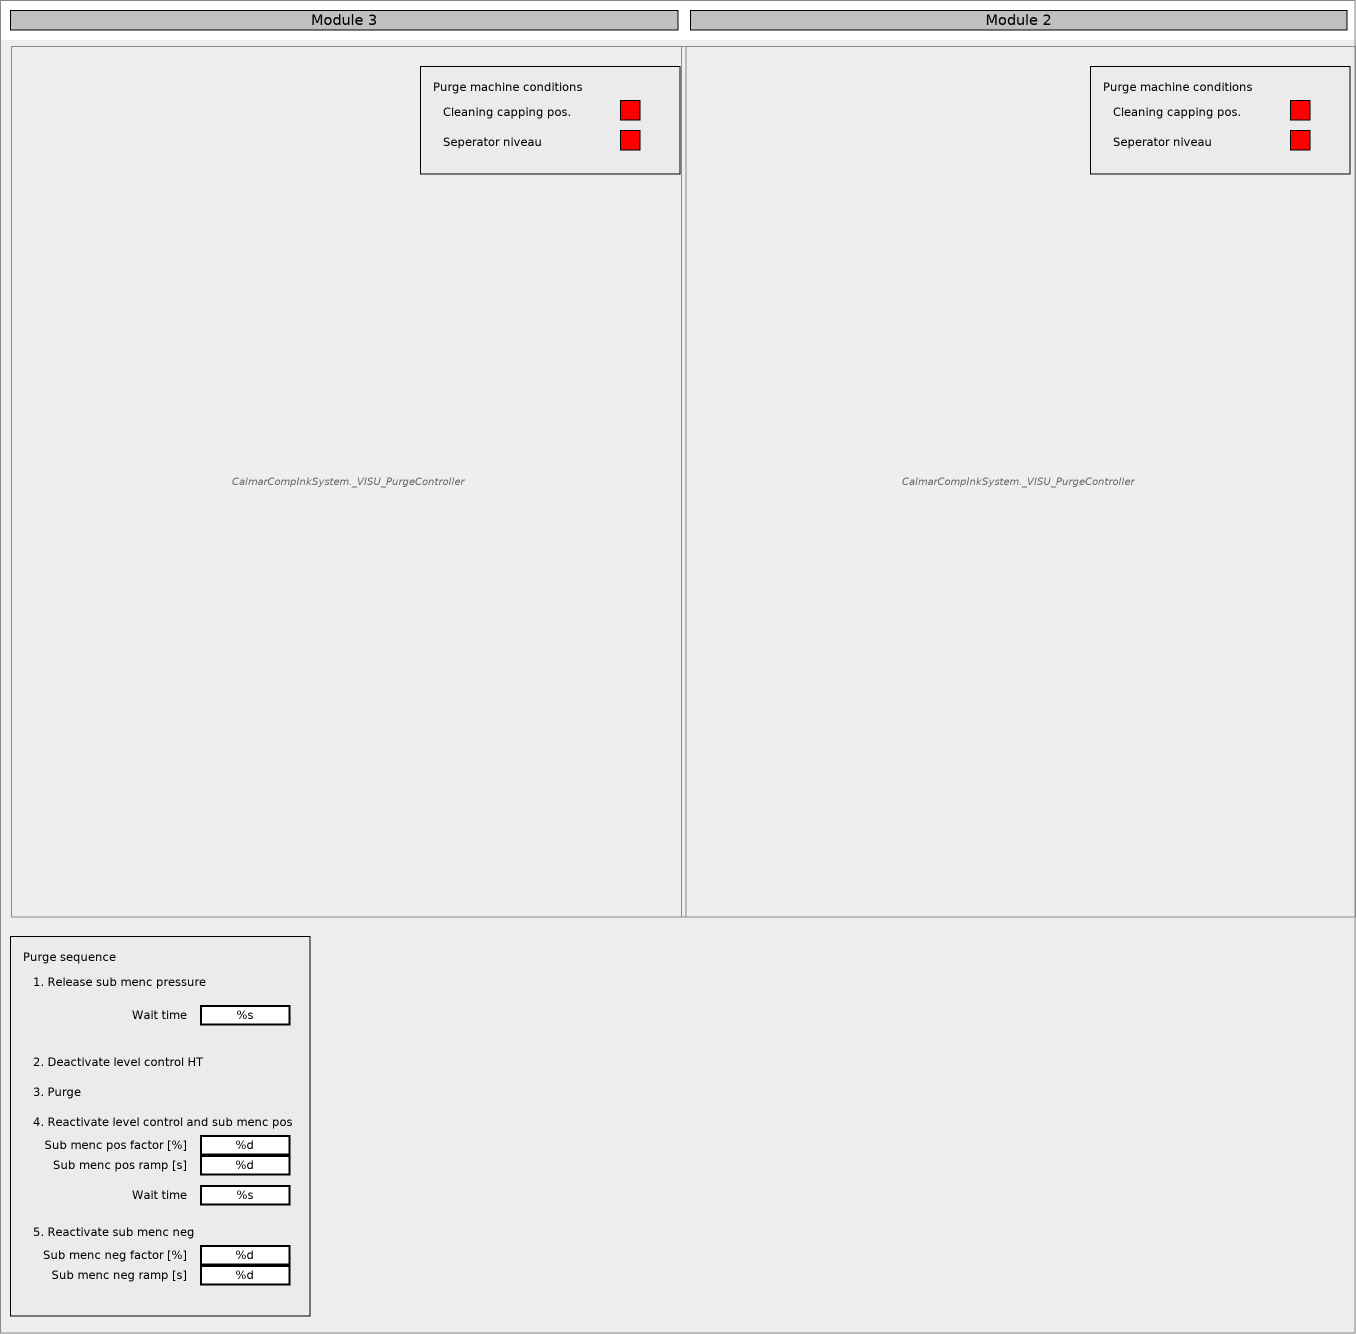
VISUALIZATION VISU_PURGE  // 1356x1334
    Rectangle (0,40 1356x1294)
    Frame (11,46 675x871)
        shows CalmarCompInkSystem._VISU_PurgeController(m_Inst_Fb := PRG_INK.fb_PurgeController[2])
    Rectangle (10,936 300x380), invisible if: (bCIk_PURGE_CONTR_SEQUENCE[1] = FALSE) and (bCIk_PURGE_CONTR_SEQUENCE[2] = FALSE)
    Rectangle (20,947 150x20), "Purge sequence", invisible if: (bCIk_PURGE_CONTR_SEQUENCE[1] = FALSE) and (bCIk_PURGE_CONTR_SEQUENCE[2] = FALSE)
    Rectangle (30,972 204x20), "1. Release sub menc pressure", invisible if: (bCIk_PURGE_CONTR_SEQUENCE[1] = FALSE) and (bCIk_PURGE_CONTR_SEQUENCE[2] = FALSE)
    Rectangle (60,1005 130x20), "Wait time", invisible if: (bCIk_PURGE_CONTR_SEQUENCE[1] = FALSE) and (bCIk_PURGE_CONTR_SEQUENCE[2] = FALSE)
    Rectangle (200,1005 90x20), "%s", text variable: PRG_INK.fb_PurgeController[1].tR_ReleaseTime, invisible if: (bCIk_PURGE_CONTR_SEQUENCE[1] = FALSE) and (bCIk_PURGE_CONTR_SEQUENCE[2] = FALSE)
        OnMouseDown: write the text variable via Edit
    Rectangle (30,1052 204x20), "2. Deactivate level control HT", invisible if: (bCIk_PURGE_CONTR_SEQUENCE[1] = FALSE) and (bCIk_PURGE_CONTR_SEQUENCE[2] = FALSE)
    Rectangle (30,1082 204x20), "3. Purge", invisible if: (bCIk_PURGE_CONTR_SEQUENCE[1] = FALSE) and (bCIk_PURGE_CONTR_SEQUENCE[2] = FALSE)
    Rectangle (30,1112 275x20), "4. Reactivate level control and sub menc pos", invisible if: (bCIk_PURGE_CONTR_SEQUENCE[1] = FALSE) and (bCIk_PURGE_CONTR_SEQUENCE[2] = FALSE)
    Rectangle (40,1135 150x20), "Sub menc pos factor [%]", invisible if: (bCIk_PURGE_CONTR_SEQUENCE[1] = FALSE) and (bCIk_PURGE_CONTR_SEQUENCE[2] = FALSE)
    Rectangle (200,1135 90x20), "%d", text variable: PRG_INK.fb_PurgeController[1].iR_SubMencPosFactor, invisible if: (bCIk_PURGE_CONTR_SEQUENCE[1] = FALSE) and (bCIk_PURGE_CONTR_SEQUENCE[2] = FALSE)
        OnMouseDown: write the text variable via Edit, min 1, max 100
    Rectangle (30,1222 250x20), "5. Reactivate sub menc neg", invisible if: (bCIk_PURGE_CONTR_SEQUENCE[1] = FALSE) and (bCIk_PURGE_CONTR_SEQUENCE[2] = FALSE)
    Rectangle (60,1185 130x20), "Wait time", invisible if: (bCIk_PURGE_CONTR_SEQUENCE[1] = FALSE) and (bCIk_PURGE_CONTR_SEQUENCE[2] = FALSE)
    Rectangle (200,1185 90x20), "%s", text variable: PRG_INK.fb_PurgeController[1].tR_SubMencReactivateTime, invisible if: (bCIk_PURGE_CONTR_SEQUENCE[1] = FALSE) and (bCIk_PURGE_CONTR_SEQUENCE[2] = FALSE)
        OnMouseDown: write the text variable via Edit
    Rectangle (40,1155 150x20), "Sub menc pos ramp [s]", invisible if: (bCIk_PURGE_CONTR_SEQUENCE[1] = FALSE) and (bCIk_PURGE_CONTR_SEQUENCE[2] = FALSE)
    Rectangle (200,1155 90x20), "%d", text variable: PRG_INK.fb_PurgeController[1].tR_SubMencPosRampTime, invisible if: (bCIk_PURGE_CONTR_SEQUENCE[1] = FALSE) and (bCIk_PURGE_CONTR_SEQUENCE[2] = FALSE)
        OnMouseDown: write the text variable via Edit
    Rectangle (40,1245 150x20), "Sub menc neg factor [%]", invisible if: (bCIk_PURGE_CONTR_SEQUENCE[1] = FALSE) and (bCIk_PURGE_CONTR_SEQUENCE[2] = FALSE)
    Rectangle (200,1245 90x20), "%d", text variable: PRG_INK.fb_PurgeController[1].iR_SubMencNegFactor, invisible if: (bCIk_PURGE_CONTR_SEQUENCE[1] = FALSE) and (bCIk_PURGE_CONTR_SEQUENCE[2] = FALSE)
        OnMouseDown: write the text variable via Edit, min 1, max 100
    Rectangle (40,1265 150x20), "Sub menc neg ramp [s]", invisible if: (bCIk_PURGE_CONTR_SEQUENCE[1] = FALSE) and (bCIk_PURGE_CONTR_SEQUENCE[2] = FALSE)
    Rectangle (200,1265 90x20), "%d", text variable: PRG_INK.fb_PurgeController[1].tR_SubMencNegRampTime, invisible if: (bCIk_PURGE_CONTR_SEQUENCE[1] = FALSE) and (bCIk_PURGE_CONTR_SEQUENCE[2] = FALSE)
        OnMouseDown: write the text variable via Edit
    Rectangle (420,66 260x108)
    Rectangle (430,77 203x20), "Purge machine conditions"
    Rectangle (440,102 148x20), "Cleaning capping pos."
    RoundedRectangle (620,100 20x20), colour toggle: PRG_MACHINE.fb_CleaningCU[2].pInPosCappingClean
    Rectangle (440,132 148x20), "Seperator niveau"
    RoundedRectangle (620,130 20x20), colour toggle: PRG_MACHINE.bIKp_SeparatorNiveau_Ok[2]
    Frame (681,46 675x871)
        shows CalmarCompInkSystem._VISU_PurgeController(m_Inst_Fb := PRG_INK.fb_PurgeController[1])
    Rectangle (1090,66 260x108)
    Rectangle (1100,77 203x20), "Purge machine conditions"
    Rectangle (1110,102 148x20), "Cleaning capping pos."
    RoundedRectangle (1290,100 20x20), colour toggle: PRG_MACHINE.fb_CleaningCU[1].pInPosCappingClean
    Rectangle (1110,132 148x20), "Seperator niveau"
    RoundedRectangle (1290,130 20x20), colour toggle: PRG_MACHINE.bIKp_SeparatorNiveau_Ok[1]
    Rectangle (10,10 668x20), "Module 3"
    Rectangle (690,10 657x20), "Module 2"
END_VISUALIZATION

// ---- VISUs/Projects/InkSystem/VISU_SETTINGS.TcVIS
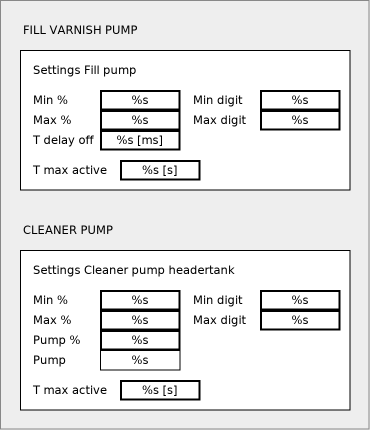
VISUALIZATION VISU_SETTINGS  // 370x430
    Rectangle (0,0 370x430)
    Rectangle (20,20 250x20), "FILL VARNISH PUMP"
    Rectangle (20,50 330x140)
    Rectangle (30,90 70x20), "Min %"
    Rectangle (30,110 70x20), "Max %"
    Rectangle (30,60 260x20), "Settings Fill pump"
    Rectangle (100,90 80x20), "%s", text variable: PRG_INK.wIDp_MinSpeedFillInkPumpVarnish
        OnMouseDown: write the text variable via Edit, min 0, max 100
    Rectangle (100,110 80x20), "%s", text variable: PRG_INK.wIDp_MaxSpeedFillInkPumpVarnish
        OnMouseDown: write the text variable via Edit, min 0, max 100
    Rectangle (100,130 80x20), "%s [ms]", text variable: PRG_INK.wIDp_PumpTimeOffDelayVarnish
        OnMouseDown: write the text variable via Edit
    Rectangle (30,130 70x20), "T delay off"
    Rectangle (190,90 70x20), "Min digit"
    Rectangle (190,110 70x20), "Max digit"
    Rectangle (260,90 80x20), "%s", text variable: PRG_INK.wIDP_AnalogMinDigitVarnish
        OnMouseDown: write the text variable via Edit, min 0, max 65535
    Rectangle (260,110 80x20), "%s", text variable: PRG_INK.wIDP_AnalogMaxDigitVarnish
        OnMouseDown: write the text variable via Edit, min 0, max 65535
    Rectangle (30,160 86x20), "T max active"
    Rectangle (120,160 80x20), "%s [s]", text variable: PRG_INK.sC_Config_I.wC_INKPUMP_MAX_TIME
        OnMouseDown: write the text variable via Edit
    Rectangle (20,220 250x20), "CLEANER PUMP"
    Rectangle (20,250 330x160)
    Rectangle (30,260 250x20), "Settings Cleaner pump headertank"
    Rectangle (30,290 70x20), "Min %"
    Rectangle (30,310 70x20), "Max %"
    Rectangle (30,350 70x20), "Pump"
    Rectangle (100,290 80x20), "%s", text variable: PRG_INK.lR_MinSpeedFillInkPumpCleaner
        OnMouseDown: write the text variable via Edit
    Rectangle (100,310 80x20), "%s", text variable: PRG_INK.lR_MaxSpeedFillInkPumpCleaner
        OnMouseDown: write the text variable via Edit
    Rectangle (100,350 80x20), "%s", text variable: PRG_INK.wL_StptSpeedCleanInkPumpDigit
    Rectangle (100,330 80x20), "%s", text variable: PRG_INK.lR_StptSpeedCleanInkPumpCleanerPercent
        OnMouseDown: write the text variable via Edit
    Rectangle (30,330 70x20), "Pump %"
    Rectangle (190,290 70x20), "Min digit"
    Rectangle (190,310 70x20), "Max digit"
    Rectangle (260,290 80x20), "%s", text variable: PRG_INK.lR_AnalogMinDigitCleaner
        OnMouseDown: write the text variable via Edit, min 0, max 65535
    Rectangle (260,310 80x20), "%s", text variable: PRG_INK.lR_AnalogMaxDigitCleaner
        OnMouseDown: write the text variable via Edit, min 0, max 65535
    Rectangle (30,380 86x20), "T max active"
    Rectangle (120,380 80x20), "%s [s]", text variable: PRG_INK.sC_Config_I.wC_CLEANERPUMP_MAX_TIME
        OnMouseDown: write the text variable via Edit
END_VISUALIZATION

// ---- VISUs/Projects/InkSystem/VISU_TEMPERATUR.TcVIS
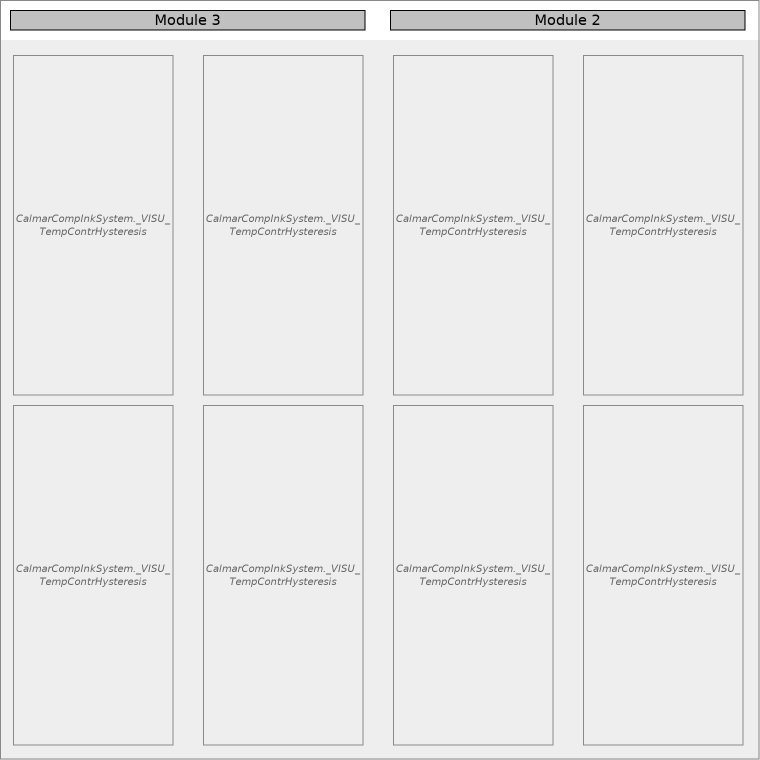
VISUALIZATION VISU_TEMPERATUR  // 760x760
    Rectangle (0,40 760x720)
    Frame (203,55 160x340)
        shows CalmarCompInkSystem._VISU_TempContrHysteresis(m_Inst_Fb := PRG_INK.fb_TempControllerHys[3])
    Frame (393,55 160x340)
        shows CalmarCompInkSystem._VISU_TempContrHysteresis(m_Inst_Fb := PRG_INK.fb_TempControllerHys[2])
    Frame (583,55 160x340)
        shows CalmarCompInkSystem._VISU_TempContrHysteresis(m_Inst_Fb := PRG_INK.fb_TempControllerHys[1])
    Frame (13,55 160x340)
        shows CalmarCompInkSystem._VISU_TempContrHysteresis(m_Inst_Fb := PRG_INK.fb_TempControllerHys[4])
    Frame (203,405 160x340)
        shows CalmarCompInkSystem._VISU_TempContrHysteresis(m_Inst_Fb := PRG_INK.fb_TempControllerHys[7])
    Frame (393,405 160x340)
        shows CalmarCompInkSystem._VISU_TempContrHysteresis(m_Inst_Fb := PRG_INK.fb_TempControllerHys[6])
    Frame (583,405 160x340)
        shows CalmarCompInkSystem._VISU_TempContrHysteresis(m_Inst_Fb := PRG_INK.fb_TempControllerHys[5])
    Frame (13,405 160x340)
        shows CalmarCompInkSystem._VISU_TempContrHysteresis(m_Inst_Fb := PRG_INK.fb_TempControllerHys[8])
    Rectangle (10,10 355x20), "Module 3"
    Rectangle (390,10 355x20), "Module 2"
END_VISUALIZATION

// ---- VISUs/Projects/InkSystem/VISU_VACUUM.TcVIS
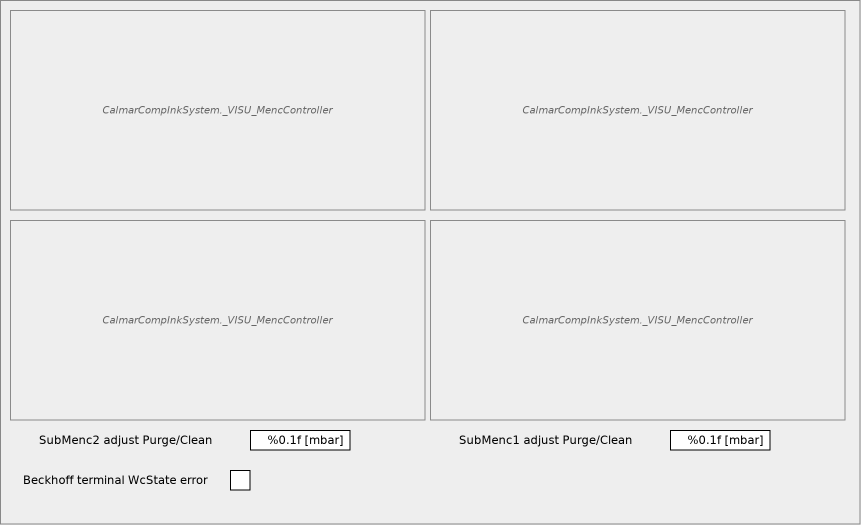
VISUALIZATION VISU_VACUUM  // 861x525
    Rectangle (0,0 861x525)
    RoundedRectangle (230,470 20x20), colour toggle: PRG_INK.bI_InkLevel1WcState
    Rectangle (20,470 200x20), "Beckhoff terminal WcState error"
    Frame (10,10 415x200)
        shows CalmarCompInkSystem._VISU_MencController(m_Inst_Fb := PRG_INK.fb_DgasMencContr[1])
    Frame (430,10 415x200)
        shows CalmarCompInkSystem._VISU_MencController(m_Inst_Fb := PRG_INK.fb_MeniscusMencContr[1])
    Frame (430,220 415x200)
        shows CalmarCompInkSystem._VISU_MencController(m_Inst_Fb := PRG_INK.fb_MeniscusMencContr[2])
    Frame (10,220 415x200)
        shows CalmarCompInkSystem._VISU_MencController(m_Inst_Fb := PRG_INK.fb_MeniscusMencContr[3])
    Rectangle (36,430 209x20), "SubMenc2 adjust Purge/Clean"
    Rectangle (250,430 100x20), "%0.1f [mbar]", text variable: PRG_INK.fR_SubMencSetAdjustWhilePurgeClean[2]
        OnMouseClick: write the text variable via Default
    Rectangle (456,430 209x20), "SubMenc1 adjust Purge/Clean"
    Rectangle (670,430 100x20), "%0.1f [mbar]", text variable: PRG_INK.fR_SubMencSetAdjustWhilePurgeClean[1]
        OnMouseClick: write the text variable via Default
END_VISUALIZATION

// ---- VISUs/Projects/Machine/Templates/_VISU_CLEAN_CH.TcVIS
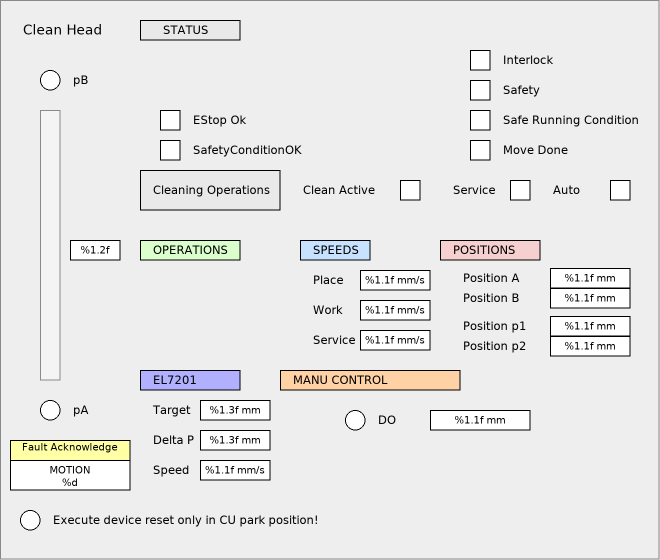
VISUALIZATION _VISU_CLEAN_CH  // 660x560
VAR_IN_OUT
  m_Inst : INT;               (*visu instance*) 
END_VAR
    Rectangle (0,0 660x560)
    Polyline (210,380)
    Polyline (510,250)
    Polyline (300,250)
    Rectangle (280,370 180x20)
    Rectangle (300,240 70x20)
    Rectangle (440,240 100x20)
    Rectangle (140,240 100x20)
    Rectangle (70,400 40x20), "pA"
    Ellipse (40,400 20x20), colour toggle: PRG_MACHINE.fb_CleaningCH[m_Inst].bL_Sensor_pA
    Ellipse (40,70 20x20), colour toggle: PRG_MACHINE.fb_CleaningCH[m_Inst].bI_Sensor_pB
    Rectangle (70,70 50x20), "pB"
    Rectangle (70,240 50x20), "%1.2f", text variable: 1000 * PRG_MACHINE.fb_CleaningCH[m_Inst].fB_Axis.fO_ActualPosition
    Rectangle (375,410 40x20), "DO"
    Rectangle (290,370 170x20), "MANU CONTROL"
    Polyline (450,380)
    Rectangle (310,240 70x20), "SPEEDS"
    Rectangle (360,270 70x20), "%1.1f mm/s", text variable: PRG_MACHINE.fb_CleaningCH[m_Inst].sI_SpeedDef.fP_PlaceSpeed
        OnMouseDown: write the text variable via VisuDialogs.Numpad
    Rectangle (360,300 70x20), "%1.1f mm/s", text variable: PRG_MACHINE.fb_CleaningCH[m_Inst].sI_SpeedDef.fP_WorkSpeed
        OnMouseDown: write the text variable via VisuDialogs.Numpad
    Rectangle (360,330 70x20), "%1.1f mm/s", text variable: PRG_MACHINE.fb_CleaningCH[m_Inst].sI_SpeedDef.fP_ServiceSpeed
        OnMouseDown: write the text variable via VisuDialogs.Numpad
    Rectangle (310,270 60x20), "Place"
    Rectangle (310,300 60x20), "Work"
    Rectangle (310,330 60x20), "Service"
        OnMouseDown: write the text variable via Edit
    Rectangle (550,268 80x20), "%1.1f mm", text variable: PRG_MACHINE.fb_CleaningCH[m_Inst].fI_Position_A
        OnMouseDown: write the text variable via VisuDialogs.Numpad
    Rectangle (460,268 85x20), "Position A"
    Rectangle (460,288 85x20), "Position B"
    Rectangle (550,288 80x20), "%1.1f mm", text variable: PRG_MACHINE.fb_CleaningCH[m_Inst].fI_Position_B
        OnMouseDown: write the text variable via VisuDialogs.Numpad
    Rectangle (450,240 90x20), "POSITIONS"
    Polyline (210,250)
    Rectangle (150,240 90x20), "OPERATIONS"
    Scrollbar (40,110 20x270)
        p3598130195: PRG_MACHINE.sADS_CleanAxis[iCPr_MAP_Cp_ChAxis[m_Inst]].sO_AxisPosition.fC_Min
        p2245068023: PRG_MACHINE.sADS_CleanAxis[iCPr_MAP_Cp_ChAxis[m_Inst]].sO_AxisPosition.fC_Max
        p1057716461: PRG_MACHINE.fb_CleaningCH[m_Inst].fB_Axis.fO_ActualPosition * 1000
    Ellipse (345,410 20x20), colour toggle: PRG_MACHINE.sADS_CleanAxis[iCPr_MAP_Cp_ChAxis[m_Inst]].bI_ManualMove, input disabled if: NOT PRG_MACHINE.sADS_CleanAxis[iCPr_MAP_Cp_ChAxis[m_Inst]].bO_ManualMoveCanEx
        toggle PRG_MACHINE.sADS_CleanAxis[iCPr_MAP_Cp_ChAxis[m_Inst]].bI_ManualMove
    Rectangle (20,20 120x20), "Clean Head"
    Rectangle (140,370 100x20)
    Rectangle (150,460 70x20), "Speed"
    Rectangle (200,460 70x20), "%1.1f mm/s", text variable: 1000 * PRG_MACHINE.fb_CleaningCH[m_Inst].fB_Axis.fI_SpeedLimit
    Rectangle (150,370 90x20), "EL7201"
    Rectangle (10,440 120x50), "Fault Acknowledge", colour toggle: (PRG_MACHINE.fb_CleaningCH[m_Inst].wL_ErrorCode) <> 0
    Polyline (130,450)
    RoundedRectangle (10,460 120x30), "%d", text variable: PRG_MACHINE.fb_CleaningCH[m_Inst].wL_ErrorCode
        tap PRG_MACHINE.sADS_CleanAxis[iCPr_MAP_Cp_ChAxis[m_Inst]].bI_FaultAck
    RoundedRectangle (40,460 60x20), "MOTION"
    Rectangle (140,170 140x40)
    Rectangle (140,20 100x20)
    Polyline (140,30)
    Polyline (240,30)
    Rectangle (160,20 60x20), "STATUS"
    RoundedRectangle (160,110 20x20), colour toggle: PRG_MACHINE.bL_IO_EStopOK
    RoundedRectangle (160,140 20x20), colour toggle: PRG_MACHINE.fB_Machine.bI_SafetyOk
    RoundedRectangle (470,140 20x20), colour toggle: NOT PRG_MACHINE.fb_CleaningCH[m_Inst].bL_Busy
    Rectangle (190,110 120x20), "EStop Ok"
    Rectangle (190,140 120x20), "SafetyConditionOK"
    Rectangle (500,140 90x20), "Move Done"
    RoundedRectangle (470,80 20x20), colour toggle: PRG_MACHINE.fb_CleaningCH[m_Inst].bI_SafeToMove
    Rectangle (500,80 120x20), "Safety"
    RoundedRectangle (470,50 20x20), colour toggle: PRG_MACHINE.fb_CleaningCH[m_Inst].bI_SafeToMove
    Rectangle (500,50 120x20), "Interlock"
    Polyline (650,160)
    Rectangle (150,180 140x20), "Cleaning Operations"
    Polyline (280,200)
    RoundedRectangle (470,110 20x20), colour toggle: PRG_MACHINE.fb_CleaningCH[m_Inst].bL_SafeRunningCondition
    Rectangle (500,110 150x20), "Safe Running Condition"
    RoundedRectangle (610,180 20x20), colour toggle: PRG_MACHINE.fb_CleanProcess[m_Inst].bI_UsrAutoMode
    Rectangle (550,180 60x20), "Auto"
    Polyline (350,80)
    RoundedRectangle (510,180 20x20), colour toggle: PRG_MACHINE.fb_CleanProcess[m_Inst].bI_UsrService
    Rectangle (450,180 60x20), "Service"
    Rectangle (300,180 90x20), "Clean Active"
    RoundedRectangle (400,180 20x20), colour toggle: PRG_MACHINE.fb_CleanProcess[m_Inst].fB_StateCleaning.bL_DevOpActive
    Rectangle (200,400 70x20), "%1.3f mm", text variable: 1000 * PRG_MACHINE.fb_CleaningCH[m_Inst].fB_Axis.fI_TargetPosition
    Rectangle (150,400 70x20), "Target"
    Rectangle (150,430 70x20), "Delta P"
    Rectangle (200,430 70x20), "%1.3f mm", text variable: 1000 * PRG_MACHINE.fb_CleaningCH[m_Inst].fB_Axis.fL_Delta_P
    Rectangle (430,410 100x20), "%1.1f mm", text variable: PRG_MACHINE.sADS_CleanAxis[iCPr_MAP_Cp_ChAxis[m_Inst]].fI_ManualTargetPos
        OnMouseDown: write the text variable via VisuDialogs.Numpad, min PRG_MACHINE.fb_CleaningCH[m_Inst].fI_Position_A, max PRG_MACHINE.fb_CleaningCH[m_Inst].fI_Position_B
    Rectangle (550,316 80x20), "%1.1f mm", text variable: PRG_MACHINE.fb_CleaningCH[m_Inst].fI_Position_p1
        OnMouseDown: write the text variable via VisuDialogs.Numpad
    Rectangle (460,316 85x20), "Position p1"
    Rectangle (460,336 85x20), "Position p2"
    Rectangle (550,336 80x20), "%1.1f mm", text variable: PRG_MACHINE.fb_CleaningCH[m_Inst].fI_Position_p2
        OnMouseDown: write the text variable via VisuDialogs.Numpad
    Ellipse (20,510 20x20), colour toggle: PRG_MACHINE.fb_CleaningCH[m_Inst].bIDp_DeviceReset, input disabled if: NOT PRG_MACHINE.fb_CleaningCU[m_Inst].pInPosCappingClean
        tap PRG_MACHINE.fb_CleaningCH[m_Inst].bIDp_DeviceReset
    Rectangle (50,510 306x20), "Execute device reset only in CU park position!"
END_VISUALIZATION

// ---- VISUs/Projects/Machine/Templates/_VISU_CLEAN_CU.TcVIS
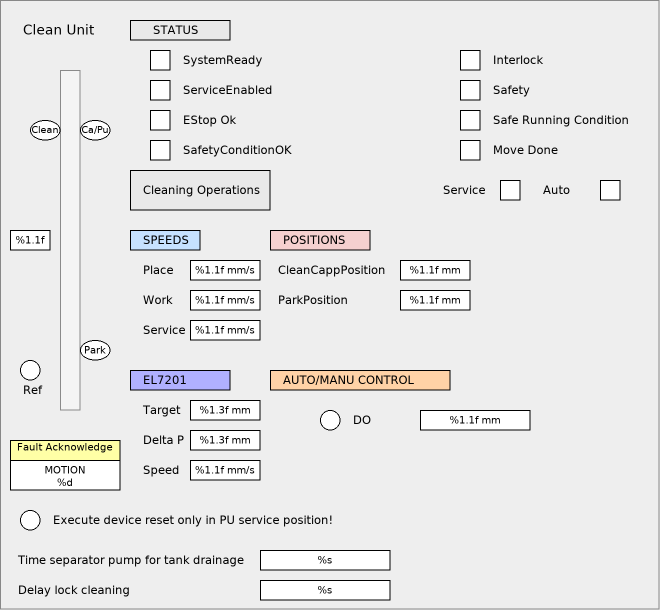
VISUALIZATION _VISU_CLEAN_CU  // 660x610
VAR_IN_OUT
  m_Inst : INT;               (*visu instance*) 
END_VAR
    Rectangle (0,0 660x610)
    Polyline (200,380)
    Rectangle (130,370 100x20)
    Rectangle (270,370 180x20)
    Rectangle (270,230 100x20)
    Rectangle (130,230 70x20)
    Rectangle (280,370 170x20), "AUTO/MANU CONTROL"
    Polyline (440,380)
    Ellipse (20,360 20x20), colour toggle: PRG_MACHINE.fb_CleaningCU[m_Inst].bL_ReferenceSensor
    Rectangle (20,380 30x20), "Ref"
    Scrollbar (60,70 20x340)
        p3598130195: -0.01
        p2245068023: 0.6
        p1057716461: PRG_MACHINE.fb_CleaningCU[m_Inst].fB_Axis.fO_ActualPosition
    Rectangle (10,230 40x20), "%1.1f", text variable: 1000 * PRG_MACHINE.fb_CleaningCU[m_Inst].fB_Axis.fO_ActualPosition
    Rectangle (140,230 70x20), "SPEEDS"
    Polyline (130,240)
    Polyline (340,240)
    Rectangle (280,230 90x20), "POSITIONS"
    Rectangle (190,400 70x20), "%1.3f mm", text variable: 1000 * PRG_MACHINE.fb_CleaningCU[m_Inst].fB_Axis.fI_TargetPosition
    Rectangle (140,400 70x20), "Target"
    Rectangle (140,460 70x20), "Speed"
    Rectangle (190,460 70x20), "%1.1f mm/s", text variable: 1000 * PRG_MACHINE.fb_CleaningCU[m_Inst].fB_Axis.fI_SpeedLimit
    Rectangle (140,370 90x20), "EL7201"
    Rectangle (140,430 70x20), "Delta P"
    Rectangle (190,430 70x20), "%1.3f mm", text variable: 1000 * PRG_MACHINE.fb_CleaningCU[m_Inst].fB_Axis.fL_Delta_P
    Ellipse (30,120 30x20), "Clean", colour toggle: PRG_MACHINE.fb_CleaningCU[m_Inst].pInPosCappingClean
    Ellipse (80,340 30x20), "Park", colour toggle: PRG_MACHINE.fb_CleaningCU[m_Inst].pInPosPark
    Ellipse (80,120 30x20), "Ca/Pu", colour toggle: PRG_MACHINE.fb_CleaningCU[m_Inst].pInPosCappingClean
    Rectangle (20,20 110x20), "Clean Unit"
    Rectangle (10,440 110x50), "Fault Acknowledge", colour toggle: (PRG_MACHINE.fb_CleaningCU[m_Inst].wL_ErrorCode) <> 0
    RoundedRectangle (10,460 110x30), "%d", text variable: PRG_MACHINE.fB_CleaningCU[m_Inst].wL_ErrorCode
        tap PRG_MACHINE.sADS_CleanAxis[iCPr_MAP_Cp_CuAxis[m_Inst]].bI_FaultAck
    RoundedRectangle (10,460 110x20), "MOTION"
    Rectangle (130,170 140x40)
    Rectangle (130,20 100x20)
    Polyline (130,30)
    Polyline (230,30)
    Rectangle (150,20 60x20), "STATUS"
    RoundedRectangle (150,80 20x20), colour toggle: PRG_MACHINE.fb_CleanProcess[m_Inst].bI_UsrService
    RoundedRectangle (150,110 20x20), colour toggle: PRG_MACHINE.bL_IO_EStopOK
    RoundedRectangle (150,140 20x20), colour toggle: PRG_MACHINE.fB_Machine.bI_SafetyOk
    RoundedRectangle (460,140 20x20), colour toggle: NOT PRG_MACHINE.fb_CleaningCU[m_Inst].bL_Busy
    RoundedRectangle (150,50 20x20), colour toggle: PRG_MACHINE.fB_Machine.bI_MachineReady
    Rectangle (180,50 120x20), "SystemReady"
    Rectangle (180,80 120x20), "ServiceEnabled"
    Rectangle (180,110 120x20), "EStop Ok"
    Rectangle (180,140 120x20), "SafetyConditionOK"
    Rectangle (490,140 90x20), "Move Done"
    RoundedRectangle (460,80 20x20), colour toggle: PRG_MACHINE.fb_CleaningCU[m_Inst].bI_SafeToMove
    Rectangle (490,80 120x20), "Safety"
    RoundedRectangle (460,50 20x20), colour toggle: PRG_MACHINE.fb_CleaningCU[m_Inst].bI_SafeToMove
    Rectangle (490,50 120x20), "Interlock"
    Polyline (640,160)
    Rectangle (140,180 140x20), "Cleaning Operations"
    Polyline (270,200)
    RoundedRectangle (460,110 20x20), colour toggle: PRG_MACHINE.fb_CleaningCU[m_Inst].bL_SafeRunningCondition
    Rectangle (490,110 150x20), "Safe Running Condition"
    RoundedRectangle (600,180 20x20), colour toggle: PRG_MACHINE.fb_CleanProcess[m_Inst].bI_UsrAutoMode
    Rectangle (540,180 60x20), "Auto"
    Polyline (340,80)
    RoundedRectangle (500,180 20x20), colour toggle: PRG_MACHINE.fb_CleanProcess[m_Inst].bI_UsrService
    Rectangle (440,180 60x20), "Service"
    Rectangle (420,410 110x20), "%1.1f mm", text variable: PRG_MACHINE.sADS_CleanAxis[iCPr_MAP_Cp_CuAxis[m_Inst]].fI_ManualTargetPos
        OnMouseDown: write the text variable via VisuDialogs.Numpad, min PRG_MACHINE.sADS_CleanAxis[iCPr_MAP_Cp_CuAxis[m_Inst]].sO_AxisPosition.fC_Min, max PRG_MACHINE.sADS_CleanAxis[iCPr_MAP_Cp_CuAxis[m_Inst]].sO_AxisPosition.fC_Max
    Rectangle (350,410 60x20), "DO"
    Ellipse (320,410 20x20), colour toggle: PRG_MACHINE.sADS_CleanAxis[iCPr_MAP_Cp_CuAxis[m_Inst]].bI_ManualMove, input disabled if: NOT PRG_MACHINE.sADS_CleanAxis[iCPr_MAP_Cp_CuAxis[m_Inst]].bO_ManualMoveCanEx
        toggle PRG_MACHINE.sADS_CleanAxis[iCPr_MAP_Cp_CuAxis[m_Inst]].bI_ManualMove
    Rectangle (190,260 70x20), "%1.1f mm/s", text variable: PRG_MACHINE.fb_CleaningCU[m_Inst].sI_SpeedDef.fP_PlaceSpeed
        OnMouseDown: write the text variable via VisuDialogs.Numpad
    Rectangle (190,290 70x20), "%1.1f mm/s", text variable: PRG_MACHINE.fb_CleaningCU[m_Inst].sI_SpeedDef.fP_WorkSpeed
        OnMouseDown: write the text variable via VisuDialogs.Numpad
    Rectangle (190,320 70x20), "%1.1f mm/s", text variable: PRG_MACHINE.fb_CleaningCU[m_Inst].sI_SpeedDef.fP_ServiceSpeed
        OnMouseDown: write the text variable via VisuDialogs.Numpad
    Rectangle (140,260 60x20), "Place"
    Rectangle (140,290 60x20), "Work"
    Rectangle (140,320 60x20), "Service"
    Rectangle (400,260 70x20), "%1.1f mm", text variable: PRG_MACHINE.fb_CleaningCU[m_Inst].fI_PositionCappingClean
        OnMouseDown: write the text variable via VisuDialogs.Numpad
    Rectangle (275,260 125x20), "CleanCappPosition"
    Rectangle (15,550 240x20), "Time separator pump for tank drainage"
    Rectangle (260,550 130x20), "%s", text variable: PRG_MACHINE.tR_TimeSeparatorPump
        OnMouseDown: write the text variable via Default
    Rectangle (400,290 70x20), "%1.1f mm", text variable: PRG_MACHINE.fb_CleaningCU[m_Inst].fI_PositionPark
        OnMouseDown: write the text variable via VisuDialogs.Numpad
    Rectangle (275,290 125x20), "ParkPosition"
    Ellipse (20,510 20x20), colour toggle: PRG_MACHINE.fb_CleaningCU[m_Inst].bIDp_DeviceReset, input disabled if: PRG_MACHINE.fb_CleaningPU[m_Inst].pInPosService
        tap PRG_MACHINE.fb_CleaningCU[m_Inst].bIDp_DeviceReset
    Rectangle (50,510 306x20), "Execute device reset only in PU service position!"
    Rectangle (15,580 240x20), "Delay lock cleaning"
    Rectangle (260,580 130x20), "%s", text variable: PRG_MACHINE.tR_TimeSeparatorLevelCheck
        OnMouseDown: write the text variable via Default
END_VISUALIZATION

// ---- VISUs/Projects/Machine/Templates/_VISU_CLEAN_PROCESS.TcVIS
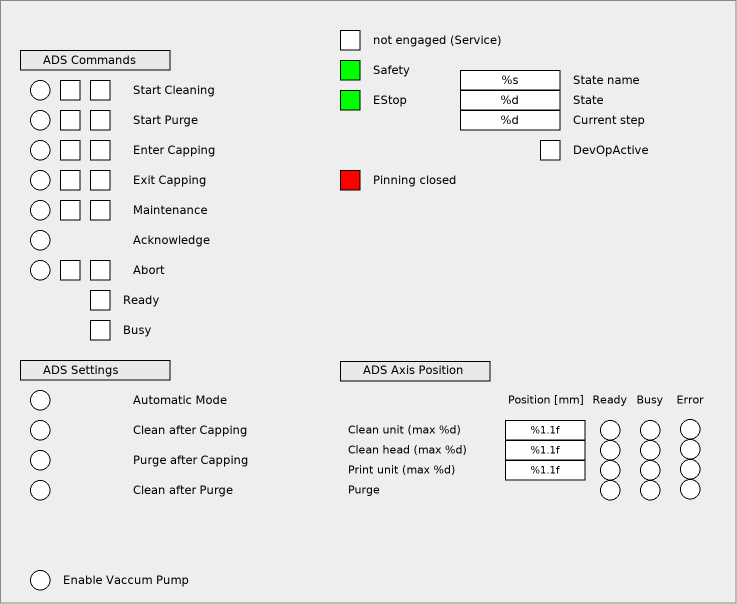
VISUALIZATION _VISU_CLEAN_PROCESS  // 737x604
VAR_IN_OUT
  m_Inst : INT;               (*visu instance*) 
END_VAR
    Rectangle (0,0 737x604)
    Polyline (20,50)
    Polyline (360,360)
    Rectangle (130,80 90x20), "Start Cleaning"
    Ellipse (30,80 20x20), colour toggle: PRG_MACHINE.sADS_CleanProcess[m_Inst].bI_Clean
        tap PRG_MACHINE.sADS_CleanProcess[m_Inst].bI_Clean
    Rectangle (130,110 90x20), "Start Purge"
    Rectangle (130,140 90x20), "Enter Capping"
    Rectangle (130,170 90x20), "Exit Capping"
    Rectangle (130,200 90x20), "Maintenance"
    RoundedRectangle (90,290 20x20), colour toggle: PRG_MACHINE.sADS_CleanProcess[m_Inst].bO_Ready
    Rectangle (120,290 120x20), "Ready"
    Rectangle (460,70 100x20), "%s", text variable: PRG_MACHINE.fb_CleanProcess[m_Inst].sL_CurrentState^.sL_StateName
    Rectangle (570,70 100x20), "State name"
    Rectangle (460,90 100x20), "%d", text variable: PRG_MACHINE.fb_CleanProcess[m_Inst].sL_CurrentState^.iL_State
    Rectangle (570,90 100x20), "State"
    Rectangle (20,50 150x20)
    Rectangle (40,50 130x20), "ADS Commands"
    RoundedRectangle (60,80 20x20), colour toggle: PRG_MACHINE.sADS_CleanProcess[m_Inst].bO_CleanCanEx
    RoundedRectangle (90,80 20x20), colour toggle: PRG_MACHINE.sADS_CleanProcess[m_Inst].bO_CleanExec
    Ellipse (30,110 20x20), colour toggle: PRG_MACHINE.sADS_CleanProcess[m_Inst].bI_Purge
        tap PRG_MACHINE.sADS_CleanProcess[m_Inst].bI_Purge
    RoundedRectangle (60,110 20x20), colour toggle: PRG_MACHINE.sADS_CleanProcess[m_Inst].bO_PurgeCanEx
    RoundedRectangle (90,110 20x20), colour toggle: PRG_MACHINE.sADS_CleanProcess[m_Inst].bO_PurgeExec
    Ellipse (30,140 20x20), colour toggle: PRG_MACHINE.sADS_CleanProcess[m_Inst].bI_StartCapping
        tap PRG_MACHINE.sADS_CleanProcess[m_Inst].bI_StartCapping
    RoundedRectangle (60,140 20x20), colour toggle: PRG_MACHINE.sADS_CleanProcess[m_Inst].bO_StartCappingCanEx
    RoundedRectangle (90,140 20x20), colour toggle: PRG_MACHINE.sADS_CleanProcess[m_Inst].bO_StartCappingExec
    Ellipse (30,170 20x20), colour toggle: PRG_MACHINE.sADS_CleanProcess[m_Inst].bI_StopCapping
        tap PRG_MACHINE.sADS_CleanProcess[m_Inst].bI_StopCapping
    RoundedRectangle (60,170 20x20), colour toggle: PRG_MACHINE.sADS_CleanProcess[m_Inst].bO_StopCappingCanEx
    RoundedRectangle (90,170 20x20), colour toggle: PRG_MACHINE.sADS_CleanProcess[m_Inst].bO_StopCappingExec
    Ellipse (30,200 20x20), colour toggle: PRG_MACHINE.sADS_CleanProcess[m_Inst].bI_Maintenance
        tap PRG_MACHINE.sADS_CleanProcess[m_Inst].bI_Maintenance
    RoundedRectangle (60,200 20x20), colour toggle: PRG_MACHINE.sADS_CleanProcess[m_Inst].bO_MaintenanceCanEx
    RoundedRectangle (90,200 20x20), colour toggle: PRG_MACHINE.sADS_CleanProcess[m_Inst].bO_MaintenanceExec
    Rectangle (130,260 90x20), "Abort"
    Ellipse (30,260 20x20), colour toggle: PRG_MACHINE.sADS_CleanProcess[m_Inst].bI_Abort
        tap PRG_MACHINE.sADS_CleanProcess[m_Inst].bI_Abort
    RoundedRectangle (60,260 20x20), colour toggle: PRG_MACHINE.sADS_CleanProcess[m_Inst].bO_AbortCanEx
    RoundedRectangle (90,260 20x20), colour toggle: PRG_MACHINE.sADS_CleanProcess[m_Inst].bO_AbortExec
    RoundedRectangle (90,320 20x20), colour toggle: PRG_MACHINE.sADS_CleanProcess[m_Inst].bO_Busy
    Rectangle (120,320 120x20), "Busy"
    Rectangle (20,360 150x20)
    Rectangle (40,360 130x20), "ADS Settings"
    Polyline (40,360)
    RoundedRectangle (340,90 20x20), colour toggle: NOT PRG_MACHINE.bL_IO_EStopOK
    Rectangle (370,30 180x20), "not engaged (Service)"
    Rectangle (505,420 80x20), "%1.1f", text variable: PRG_MACHINE.sADS_CleanAxis[iCPr_MAP_Cp_CuAxis[m_Inst]].sO_AxisPosition.fO_Val
    Rectangle (505,440 80x20), "%1.1f", text variable: PRG_MACHINE.sADS_CleanAxis[iCPr_MAP_Cp_ChAxis[m_Inst]].sO_AxisPosition.fO_Val
    Rectangle (505,460 80x20), "%1.1f", text variable: PRG_MACHINE.sADS_CleanAxis[iCPr_MAP_Cp_PuAxis[m_Inst]].sO_AxisPosition.fO_Val
    Ellipse (600,420 20x20), colour toggle: PRG_MACHINE.sADS_CleanAxis[iCPr_MAP_Cp_CuAxis[m_Inst]].bO_Ready
    Ellipse (640,420 20x20), colour toggle: PRG_MACHINE.sADS_CleanAxis[iCPr_MAP_Cp_CuAxis[m_Inst]].bO_Busy
    Ellipse (600,440 20x20), colour toggle: PRG_MACHINE.sADS_CleanAxis[iCPr_MAP_Cp_ChAxis[m_Inst]].bO_Ready
    Ellipse (640,440 20x20), colour toggle: PRG_MACHINE.sADS_CleanAxis[iCPr_MAP_Cp_ChAxis[m_Inst]].bO_Busy
    Ellipse (600,460 20x20), colour toggle: PRG_MACHINE.sADS_CleanAxis[iCPr_MAP_Cp_PuAxis[m_Inst]].bO_Ready
    Ellipse (640,460 20x20), colour toggle: PRG_MACHINE.sADS_CleanAxis[iCPr_MAP_Cp_PuAxis[m_Inst]].bO_Busy
    Rectangle (590,390 40x20), "Ready"
    Rectangle (630,390 40x20), "Busy"
    Rectangle (505,390 83x20), "Position [mm]"
    Rectangle (340,361 150x20)
    Rectangle (360,360 130x20), "ADS Axis Position"
    Ellipse (600,480 20x20), colour toggle: PRG_MACHINE.sADS_CleanAxis[iCPr_MAP_Cp_InkInterface[m_Inst]].bO_Ready
    Ellipse (640,480 20x20), colour toggle: PRG_MACHINE.sADS_CleanAxis[iCPr_MAP_Cp_InkInterface[m_Inst]].bO_Busy
    Rectangle (345,480 150x20), "Purge"
    Ellipse (680,419 20x20), colour toggle: PRG_MACHINE.sADS_CleanAxis[iCPr_MAP_Cp_CuAxis[m_Inst]].bO_Error
        toggle PRG_MACHINE.sADS_CleanAxis[iCPr_MAP_Cp_CuAxis[m_Inst]].bI_FaultAck
    Ellipse (680,439 20x20), colour toggle: PRG_MACHINE.sADS_CleanAxis[iCPr_MAP_Cp_ChAxis[m_Inst]].bO_Error
        toggle PRG_MACHINE.sADS_CleanAxis[iCPr_MAP_Cp_ChAxis[m_Inst]].bI_FaultAck
    Ellipse (680,459 20x20), colour toggle: PRG_MACHINE.sADS_CleanAxis[iCPr_MAP_Cp_PuAxis[m_Inst]].bO_Error
        tap PRG_MACHINE.sADS_CleanAxis[iCPr_MAP_Cp_PuAxis[m_Inst]].bI_FaultAck
    Rectangle (670,390 40x20), "Error"
    Ellipse (680,479 20x20), colour toggle: PRG_MACHINE.sADS_CleanAxis[iCPr_MAP_Cp_InkInterface[m_Inst]].bO_Error
    RoundedRectangle (340,60 20x20), colour toggle: NOT PRG_MACHINE.bL_SafetyOk[m_Inst]
    RoundedRectangle (340,30 20x20), colour toggle: PRG_MACHINE.fb_CleanProcess[m_Inst].bI_UsrService
    Rectangle (370,60 80x20), "Safety"
    Rectangle (370,90 80x20), "EStop"
    Rectangle (345,420 150x20), "Clean unit (max %d)", text variable: PRG_MACHINE.sADS_CleanAxis[iCPr_MAP_Cp_CuAxis[m_Inst]].sO_AxisPosition.fC_Max
    Rectangle (345,440 150x20), "Clean head (max %d)", text variable: PRG_MACHINE.sADS_CleanAxis[iCPr_MAP_Cp_ChAxis[m_Inst]].sO_AxisPosition.fC_Max
    Rectangle (345,460 150x20), "Print unit (max %d)", text variable: PRG_MACHINE.sADS_CleanAxis[iCPr_MAP_Cp_PuAxis[m_Inst]].sO_AxisPosition.fC_Max
    Rectangle (460,110 100x20), "%d", text variable: PRG_MACHINE.fb_CleanProcess[m_Inst].sL_CurrentState^.iL_State
    Rectangle (570,110 100x20), "Current step"
    RoundedRectangle (540,140 20x20), colour toggle: PRG_MACHINE.fb_CleanProcess[m_Inst].sL_CurrentState^.bL_DevOpActive
    Rectangle (570,140 100x20), "DevOpActive"
    Rectangle (130,390 103x20), "Automatic Mode"
    Ellipse (30,390 20x20), colour toggle: PRG_MACHINE.sADS_CleanProcess[m_Inst].bI_AutoMode
        toggle PRG_MACHINE.sADS_CleanProcess[m_Inst].bI_AutoMode
    Rectangle (130,420 150x20), "Clean after Capping"
    Ellipse (30,420 20x20), colour toggle: PRG_MACHINE.sADS_CleanProcess[m_Inst].bI_CleanAfterCapp
        toggle PRG_MACHINE.sADS_CleanProcess[m_Inst].bI_CleanAfterCapp
    Rectangle (130,480 150x20), "Clean after Purge"
    Ellipse (30,480 20x20), colour toggle: PRG_MACHINE.sADS_CleanProcess[m_Inst].bI_CleanAfterPurge
        toggle PRG_MACHINE.sADS_CleanProcess[m_Inst].bI_CleanAfterPurge
    Rectangle (130,450 150x20), "Purge after Capping"
    Ellipse (30,450 20x20), colour toggle: PRG_MACHINE.sADS_CleanProcess[m_Inst].bI_PurgeAfterCapp
        toggle PRG_MACHINE.sADS_CleanProcess[m_Inst].bI_PurgeAfterCapp
    Ellipse (30,570 20x20), colour toggle: PRG_MACHINE.bL_ManualVacuumBin[m_Inst]
        toggle PRG_MACHINE.bL_ManualVacuumBin[m_Inst]
    Rectangle (60,570 138x20), "Enable Vaccum Pump"
    RoundedRectangle (340,170 20x20), colour toggle: PRG_MACHINE.IbEAP_PinningClosed[m_Inst]
    Rectangle (370,170 150x20), "Pinning closed"
    Rectangle (130,230 90x20), "Acknowledge"
    Ellipse (30,230 20x20), colour toggle: PRG_MACHINE.sADS_CleanProcess[m_Inst].bI_Maintenance
        tap PRG_MACHINE.sADS_CleanProcess[m_Inst].bI_AcknowledgeError
END_VISUALIZATION

// ---- VISUs/Projects/Machine/Templates/_VISU_CLEAN_PU.TcVIS
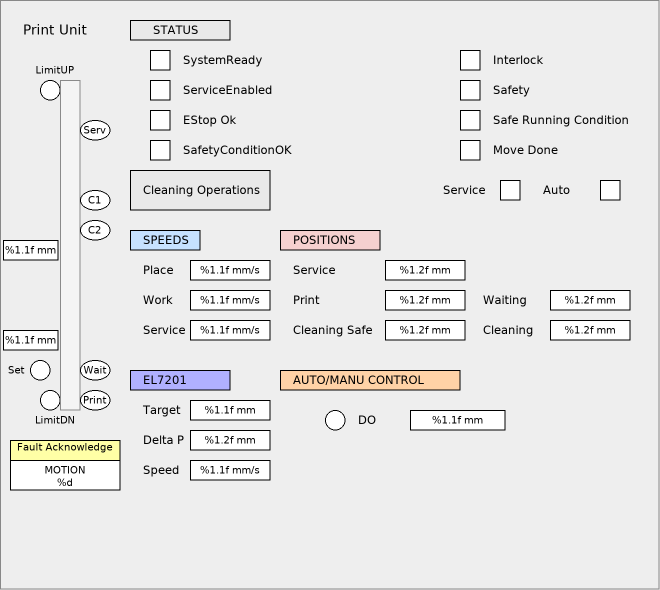
VISUALIZATION _VISU_CLEAN_PU  // 660x590
VAR_IN_OUT
  m_Inst : INT;               (*visu instance*) 
END_VAR
    Rectangle (0,0 660x590)
    Polyline (200,380)
    Polyline (130,240)
    Rectangle (130,170 140x40)
    Rectangle (130,370 100x20)
    Rectangle (280,370 180x20)
    Rectangle (280,230 100x20)
    Rectangle (130,230 70x20)
    Rectangle (130,20 100x20)
    Rectangle (20,20 100x20), "Print Unit"
    Polyline (130,30)
    Polyline (230,30)
    Rectangle (150,20 60x20), "STATUS"
    RoundedRectangle (150,80 20x20), colour toggle: PRG_MACHINE.fb_CleanProcess[m_Inst].bI_UsrService
    RoundedRectangle (150,110 20x20), colour toggle: PRG_MACHINE.bL_IO_EStopOK
    RoundedRectangle (150,140 20x20), colour toggle: PRG_MACHINE.fB_Machine.bI_SafetyOk
    RoundedRectangle (460,140 20x20), colour toggle: NOT PRG_MACHINE.fb_CleaningPU[m_Inst].bL_Busy
    RoundedRectangle (150,50 20x20), colour toggle: PRG_MACHINE.fB_Machine.bI_MachineReady
    Rectangle (180,50 120x20), "SystemReady"
    Rectangle (180,80 120x20), "ServiceEnabled"
    Rectangle (180,110 120x20), "EStop Ok"
    Rectangle (180,140 120x20), "SafetyConditionOK"
    Rectangle (490,140 90x20), "Move Done"
    Rectangle (290,370 170x20), "AUTO/MANU CONTROL"
    Polyline (450,380)
    Rectangle (30,60 50x20), "LimitUP"
    Ellipse (40,80 20x20), colour toggle: NOT PRG_MACHINE.fb_CleaningPU[m_Inst].bI_SensorTop
    Ellipse (40,390 20x20), colour toggle: NOT PRG_MACHINE.fb_CleaningPU[m_Inst].bI_SensorBottom
    Rectangle (30,410 50x20), "LimitDN"
    Scrollbar (60,80 20x330)
        p2245068023: 0.5
        p1057716461: PRG_MACHINE.fb_CleaningPU[m_Inst].fB_Axis.fO_ActualPosition
    Rectangle (140,230 70x20), "SPEEDS"
    Rectangle (190,260 80x20), "%1.1f mm/s", text variable: PRG_MACHINE.fb_CleaningPU[m_Inst].sI_SpeedDef.fP_PlaceSpeed
        OnMouseDown: write the text variable via VisuDialogs.Numpad
    Rectangle (190,290 80x20), "%1.1f mm/s", text variable: PRG_MACHINE.fb_CleaningPU[m_Inst].sI_SpeedDef.fP_WorkSpeed
        OnMouseDown: write the text variable via VisuDialogs.Numpad
    Rectangle (190,320 80x20), "%1.1f mm/s", text variable: PRG_MACHINE.fb_CleaningPU[m_Inst].sI_SpeedDef.fP_ServiceSpeed
        OnMouseDown: write the text variable via VisuDialogs.Numpad
    Rectangle (140,260 45x20), "Place"
    Rectangle (140,290 45x20), "Work"
    Rectangle (140,320 45x20), "Service"
        OnMouseDown: write the text variable via Edit
    Rectangle (290,260 90x20), "Service"
    Rectangle (290,290 90x20), "Print"
    Polyline (350,240)
    Rectangle (290,230 90x20), "POSITIONS"
    Rectangle (190,400 80x20), "%1.1f mm", text variable: 1000 * PRG_MACHINE.fb_CleaningPU[m_Inst].fB_Axis.fI_TargetPosition
    RoundedRectangle (460,80 20x20), colour toggle: PRG_MACHINE.fb_CleaningPU[m_Inst].bI_SafeToMove
    Rectangle (490,80 120x20), "Safety"
    RoundedRectangle (460,50 20x20), colour toggle: PRG_MACHINE.fb_CleaningPU[m_Inst].bI_SafeToMove
    Rectangle (490,50 120x20), "Interlock"
    Rectangle (5,360 25x20), "Set"
    Ellipse (30,360 20x20), colour toggle: PRG_MACHINE.fb_CleaningPU[m_Inst].fB_Axis.bI_SetPosition
        toggle PRG_MACHINE.fb_CleaningPU[m_Inst].fB_Axis.bI_SetPosition
    Rectangle (3,240 55x20), "%1.1f mm", text variable: 1000 * PRG_MACHINE.fb_CleaningPU[m_Inst].fB_Axis.fO_ActualPosition, colour toggle: PRG_MACHINE.fb_CleaningCH[1].bL_Sensor_pA
    Rectangle (290,320 90x20), "Cleaning Safe"
    Rectangle (385,320 80x20), "%1.2f mm", text variable: PRG_MACHINE.fb_CleaningPU[m_Inst].fI_PositionClean1
        OnMouseDown: write the text variable via VisuDialogs.Numpad
    Rectangle (140,400 45x20), "Target"
    Rectangle (140,460 45x20), "Speed"
    Rectangle (190,460 80x20), "%1.1f mm/s", text variable: 1000 * PRG_MACHINE.fb_CleaningPU[m_Inst].fB_Axis.fI_SpeedLimit
    Rectangle (140,370 90x20), "EL7201"
    Rectangle (140,430 45x20), "Delta P"
    Rectangle (190,430 80x20), "%1.2f mm", text variable: 1000 * PRG_MACHINE.fb_CleaningPU[m_Inst].fB_Axis.fL_Delta_P
    Ellipse (80,120 30x20), "Serv", colour toggle: PRG_MACHINE.fb_CleaningPU[m_Inst].pInPosService
    Ellipse (80,220 30x20), "C2", colour toggle: PRG_MACHINE.fb_CleaningPU[m_Inst].pInPosClean2
    Ellipse (80,190 30x20), "C1", colour toggle: PRG_MACHINE.fb_CleaningPU[m_Inst].pInPosClean1
    Ellipse (80,360 30x20), "Wait", colour toggle: PRG_MACHINE.fb_CleaningPU[m_Inst].pInPosWait
    Ellipse (80,390 30x20), "Print", colour toggle: PRG_MACHINE.fb_CleaningPU[m_Inst].pInPosPrint
    Polyline (640,160)
    Rectangle (140,180 140x20), "Cleaning Operations"
    Polyline (270,200)
    RoundedRectangle (460,110 20x20), colour toggle: PRG_MACHINE.fb_CleaningPU[m_Inst].bL_SafeRunningCondition
    Rectangle (490,110 140x20), "Safe Running Condition"
    RoundedRectangle (600,180 20x20), colour toggle: PRG_MACHINE.fb_CleanProcess[m_Inst].bI_UsrAutoMode
    Rectangle (540,180 55x20), "Auto"
    Polyline (340,80)
    Rectangle (10,440 110x50), "Fault Acknowledge", colour toggle: (PRG_MACHINE.fb_CleaningPU[m_Inst].wL_ErrorCode) <> 0
    RoundedRectangle (10,460 110x30), "%d", text variable: PRG_MACHINE.fb_CleaningPU[m_Inst].wL_ErrorCode
        tap PRG_MACHINE.sADS_CleanAxis[iCPr_MAP_Cp_PuAxis[m_Inst]].bI_FaultAck
    RoundedRectangle (10,460 110x20), "MOTION"
    Rectangle (3,330 55x20), "%1.1f mm", text variable: PRG_MACHINE.fb_CleaningPU[m_Inst].fL_SetPositionValue
        OnMouseDown: write the text variable via VisuDialogs.Numpad
    Rectangle (480,320 65x20), "Cleaning"
    Rectangle (550,320 80x20), "%1.2f mm", text variable: PRG_MACHINE.fb_CleaningPU[m_Inst].fI_PositionClean2
        OnMouseDown: write the text variable via VisuDialogs.Numpad
    RoundedRectangle (500,180 20x20), colour toggle: PRG_MACHINE.fb_CleanProcess[m_Inst].bI_UsrService
    Rectangle (440,180 55x20), "Service"
    Rectangle (410,410 95x20), "%1.1f mm", text variable: PRG_MACHINE.sADS_CleanAxis[iCPr_MAP_Cp_PuAxis[m_Inst]].fI_ManualTargetPos
        OnMouseDown: write the text variable via VisuDialogs.Numpad, min PRG_MACHINE.sADS_CleanAxis[iCPr_MAP_Cp_PuAxis[m_Inst]].sO_AxisPosition.fC_Min, max PRG_MACHINE.sADS_CleanAxis[iCPr_MAP_Cp_PuAxis[m_Inst]].sO_AxisPosition.fC_Max
    Rectangle (355,410 50x20), "DO"
    Ellipse (325,410 20x20), colour toggle: PRG_MACHINE.sADS_CleanAxis[iCPr_MAP_Cp_PuAxis[m_Inst]].bI_ManualMove, input disabled if: NOT PRG_MACHINE.sADS_CleanAxis[iCPr_MAP_Cp_PuAxis[m_Inst]].bO_ManualMoveCanEx
        toggle PRG_MACHINE.sADS_CleanAxis[iCPr_MAP_Cp_PuAxis[m_Inst]].bI_ManualMove
    Rectangle (385,260 80x20), "%1.2f mm", text variable: PRG_MACHINE.fb_CleaningPU[m_Inst].fI_PositionService
        OnMouseDown: write the text variable via VisuDialogs.Numpad
    Rectangle (385,290 80x20), "%1.2f mm", text variable: PRG_MACHINE.fb_CleaningPU[m_Inst].fL_PrintPositionMM
        OnMouseDown: write the text variable via VisuDialogs.Numpad, min PRG_PRINT.sAdsSheetAlignment[1].sI_HeadGap.fC_Min, max PRG_PRINT.sAdsSheetAlignment[1].sI_HeadGap.fC_Max
    Rectangle (480,290 65x20), "Waiting"
    Rectangle (550,290 80x20), "%1.2f mm", text variable: PRG_MACHINE.fb_CleaningPU[m_Inst].fI_PositionWait
        OnMouseDown: write the text variable via VisuDialogs.Numpad
END_VISUALIZATION

// ---- VISUs/Projects/Machine/VISU_EAP_MACHINE.TcVIS
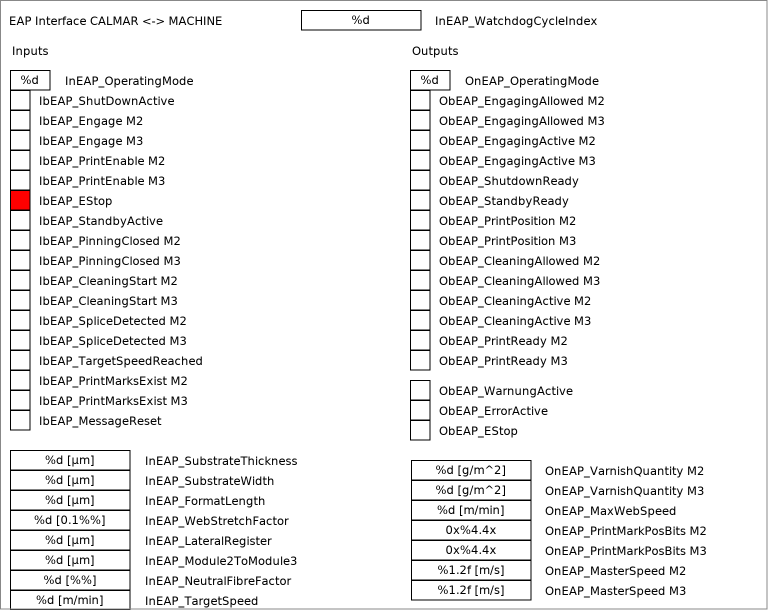
VISUALIZATION VISU_EAP_MACHINE  // 768x610
    RoundedRectangle (10,90 20x20), colour toggle: PRG_MACHINE.IbEAP_ShutDownActive
    RoundedRectangle (10,110 20x20), colour toggle: PRG_MACHINE.IbEAP_Engaged[1]
    RoundedRectangle (10,150 20x20), colour toggle: PRG_MACHINE.IbEAP_PrintEnabled[1]
    Rectangle (36,92 257x18), "IbEAP_ShutDownActive"
    Rectangle (36,112 256x18), "IbEAP_Engage M2"
    Rectangle (36,152 226x18), "IbEAP_PrintEnable M2"
    RoundedRectangle (10,190 20x20), colour toggle: NOT PRG_MACHINE.IbEAP_EStop
    Rectangle (36,192 226x18), "IbEAP_EStop"
    RoundedRectangle (10,210 20x20), colour toggle: PRG_MACHINE.IbEAP_StandbyActive
    Rectangle (36,212 226x18), "IbEAP_StandbyActive"
    RoundedRectangle (10,410 20x20), colour toggle: PRG_MACHINE.IbEAP_MessageReset
    Rectangle (36,412 226x18), "IbEAP_MessageReset"
    RoundedRectangle (10,230 20x20), colour toggle: PRG_MACHINE.IbEAP_PinningClosed[1]
    Rectangle (36,232 226x18), "IbEAP_PinningClosed M2"
    Rectangle (10,530 120x20), "%d [µm]", text variable: PRG_MACHINE.InEAP_LateralRegister
    Rectangle (142,532 226x18), "InEAP_LateralRegister"
    Rectangle (10,450 120x20), "%d [µm]", text variable: PRG_MACHINE.InEAP_SubstrateThickness
    Rectangle (142,452 226x18), "InEAP_SubstrateThickness"
    Rectangle (10,470 120x20), "%d [µm]", text variable: PRG_MACHINE.InEAP_SubstrateWidth
    Rectangle (142,472 226x18), "InEAP_SubstrateWidth"
    Rectangle (10,490 120x20), "%d [µm]", text variable: PRG_MACHINE.InEAP_FormatLength
    Rectangle (142,492 226x18), "InEAP_FormatLength"
    Rectangle (6,12 257x18), "EAP Interface CALMAR <-> MACHINE"
    RoundedRectangle (410,90 20x20), colour toggle: PRG_MACHINE.ObEAP_EngagingAllowed[1]
    Rectangle (436,92 257x18), "ObEAP_EngagingAllowed M2"
    RoundedRectangle (410,170 20x20), colour toggle: PRG_MACHINE.ObEAP_ShutdownReady
    Rectangle (436,172 257x18), "ObEAP_ShutdownReady"
    RoundedRectangle (410,190 20x20), colour toggle: PRG_MACHINE.ObEAP_StandbyReady
    Rectangle (436,192 257x18), "ObEAP_StandbyReady"
    RoundedRectangle (410,210 20x20), colour toggle: PRG_MACHINE.ObEAP_PrintPosition[1]
    Rectangle (436,212 257x18), "ObEAP_PrintPosition M2"
    Rectangle (9,42 257x18), "Inputs"
    Rectangle (409,42 257x18), "Outputs"
    Rectangle (411,480 120x20), "%d [g/m^2]", text variable: PRG_MACHINE.OnEAP_VarnishQuantity[2]
    Rectangle (542,482 226x18), "OnEAP_VarnishQuantity M3"
    Rectangle (411,500 120x20), "%d [m/min]", text variable: PRG_MACHINE.OnEAP_MaxWebSpeed
    Rectangle (542,502 226x18), "OnEAP_MaxWebSpeed"
    Rectangle (301,10 120x20), "%d", text variable: PRG_MACHINE.InEAP_WatchdogCycleIndex
    Rectangle (432,12 226x18), "InEAP_WatchdogCycleIndex"
    RoundedRectangle (410,380 20x20), colour toggle: PRG_MACHINE.ObEAP_WarnungActive
    Rectangle (436,382 257x18), "ObEAP_WarnungActive"
    RoundedRectangle (410,400 20x20), colour toggle: PRG_MACHINE.ObEAP_ErrorActive
    Rectangle (436,402 257x18), "ObEAP_ErrorActive"
    RoundedRectangle (10,270 20x20), colour toggle: PRG_MACHINE.IbEAP_CleaningStart[1]
    Rectangle (36,272 226x18), "IbEAP_CleaningStart M2"
    RoundedRectangle (410,250 20x20), colour toggle: PRG_MACHINE.ObEAP_CleaningAllowed[1]
    Rectangle (436,252 257x18), "ObEAP_CleaningAllowed M2"
    RoundedRectangle (410,310 20x20), colour toggle: PRG_MACHINE.ObEAP_CleaningActive[2]
    Rectangle (436,312 257x18), "ObEAP_CleaningActive M3"
    RoundedRectangle (410,330 20x20), colour toggle: PRG_MACHINE.ObEAP_PrintReady[1]
    Rectangle (436,332 257x18), "ObEAP_PrintReady M2"
    Rectangle (10,510 120x20), "%d [0.1%%]", text variable: PRG_MACHINE.InEAP_WebStretchFactor
    Rectangle (142,512 226x18), "InEAP_WebStretchFactor"
    Rectangle (410,70 40x20), "%d", text variable: PRG_MACHINE.OnEAP_OperatingMode
    Rectangle (462,72 171x18), "OnEAP_OperatingMode"
    Rectangle (10,70 40x20), "%d", text variable: PRG_MACHINE.InEAP_OperatingMode
    Rectangle (62,72 171x18), "InEAP_OperatingMode"
    RoundedRectangle (10,130 20x20), colour toggle: PRG_MACHINE.IbEAP_Engaged[2]
    Rectangle (36,132 256x18), "IbEAP_Engage M3"
    RoundedRectangle (10,170 20x20), colour toggle: PRG_MACHINE.IbEAP_PrintEnabled[2]
    Rectangle (36,172 226x18), "IbEAP_PrintEnable M3"
    RoundedRectangle (10,290 20x20), colour toggle: PRG_MACHINE.IbEAP_CleaningStart[2]
    Rectangle (36,292 226x18), "IbEAP_CleaningStart M3"
    RoundedRectangle (10,250 20x20), colour toggle: PRG_MACHINE.IbEAP_PinningClosed[2]
    Rectangle (36,252 226x18), "IbEAP_PinningClosed M3"
    RoundedRectangle (410,110 20x20), colour toggle: PRG_MACHINE.ObEAP_EngagingAllowed[2]
    Rectangle (436,112 257x18), "ObEAP_EngagingAllowed M3"
    RoundedRectangle (410,130 20x20), colour toggle: PRG_MACHINE.ObEAP_EngagingActive[1]
    Rectangle (436,132 257x18), "ObEAP_EngagingActive M2"
    RoundedRectangle (410,150 20x20), colour toggle: PRG_MACHINE.ObEAP_EngagingActive[2]
    Rectangle (436,152 257x18), "ObEAP_EngagingActive M3"
    RoundedRectangle (410,230 20x20), colour toggle: PRG_MACHINE.ObEAP_PrintPosition[2]
    Rectangle (436,232 257x18), "ObEAP_PrintPosition M3"
    RoundedRectangle (410,270 20x20), colour toggle: PRG_MACHINE.ObEAP_CleaningAllowed[2]
    Rectangle (436,272 257x18), "ObEAP_CleaningAllowed M3"
    RoundedRectangle (410,290 20x20), colour toggle: PRG_MACHINE.ObEAP_CleaningActive[1]
    Rectangle (436,292 257x18), "ObEAP_CleaningActive M2"
    RoundedRectangle (410,350 20x20), colour toggle: PRG_MACHINE.ObEAP_PrintReady[2]
    Rectangle (436,352 257x18), "ObEAP_PrintReady M3"
    Rectangle (411,460 120x20), "%d [g/m^2]", text variable: PRG_MACHINE.OnEAP_VarnishQuantity[1]
    Rectangle (542,462 226x18), "OnEAP_VarnishQuantity M2"
    RoundedRectangle (10,310 20x20), colour toggle: PRG_MACHINE.IbEAP_SpliceDetected[1]
    Rectangle (36,312 226x18), "IbEAP_SpliceDetected M2"
    RoundedRectangle (10,330 20x20), colour toggle: PRG_MACHINE.IbEAP_SpliceDetected[2]
    Rectangle (36,332 226x18), "IbEAP_SpliceDetected M3"
    Rectangle (10,550 120x20), "%d [µm]", text variable: PRG_MACHINE.InEAP_Module2ToModule3
    Rectangle (142,552 226x18), "InEAP_Module2ToModule3"
    RoundedRectangle (10,350 20x20), colour toggle: PRG_MACHINE.IbEAP_TargetSpeedReached]
    Rectangle (36,352 226x18), "IbEAP_TargetSpeedReached"
    RoundedRectangle (10,370 20x20), colour toggle: PRG_MACHINE.IbEAP_PrintMarksExist[1]
    Rectangle (36,372 226x18), "IbEAP_PrintMarksExist M2"
    RoundedRectangle (10,390 20x20), colour toggle: PRG_MACHINE.IbEAP_PrintMarksExist[2]
    Rectangle (36,392 226x18), "IbEAP_PrintMarksExist M3"
    Rectangle (10,570 120x20), "%d [%%]", text variable: PRG_MACHINE.InEAP_NeutralFibreFactor
    Rectangle (142,572 226x18), "InEAP_NeutralFibreFactor"
    Rectangle (10,590 120x20), "%d [m/min]", text variable: PRG_MACHINE.InEAP_NeutralFibreFactor
    Rectangle (142,592 226x18), "InEAP_TargetSpeed"
    RoundedRectangle (410,420 20x20), colour toggle: PRG_MACHINE.ObEAP_ErrorActive
    Rectangle (436,422 257x18), "ObEAP_EStop"
    Rectangle (411,540 120x20), "0x%4.4x", text variable: PRG_MACHINE.OnEAP_PrintMarkPosBits[2]
    Rectangle (542,542 226x18), "OnEAP_PrintMarkPosBits M3"
    Rectangle (411,520 120x20), "0x%4.4x", text variable: PRG_MACHINE.OnEAP_PrintMarkPosBits[1]
    Rectangle (542,522 226x18), "OnEAP_PrintMarkPosBits M2"
    Rectangle (411,580 120x20), "%1.2f [m/s]", text variable: PRG_MACHINE.OnEAP_MasterSpeed[2]
    Rectangle (542,582 226x18), "OnEAP_MasterSpeed M3"
    Rectangle (411,560 120x20), "%1.2f [m/s]", text variable: PRG_MACHINE.OnEAP_MasterSpeed[1]
    Rectangle (542,562 226x18), "OnEAP_MasterSpeed M2"
END_VISUALIZATION

// ---- VISUs/Projects/Machine/VISU_CLEAN_CH.TcVIS
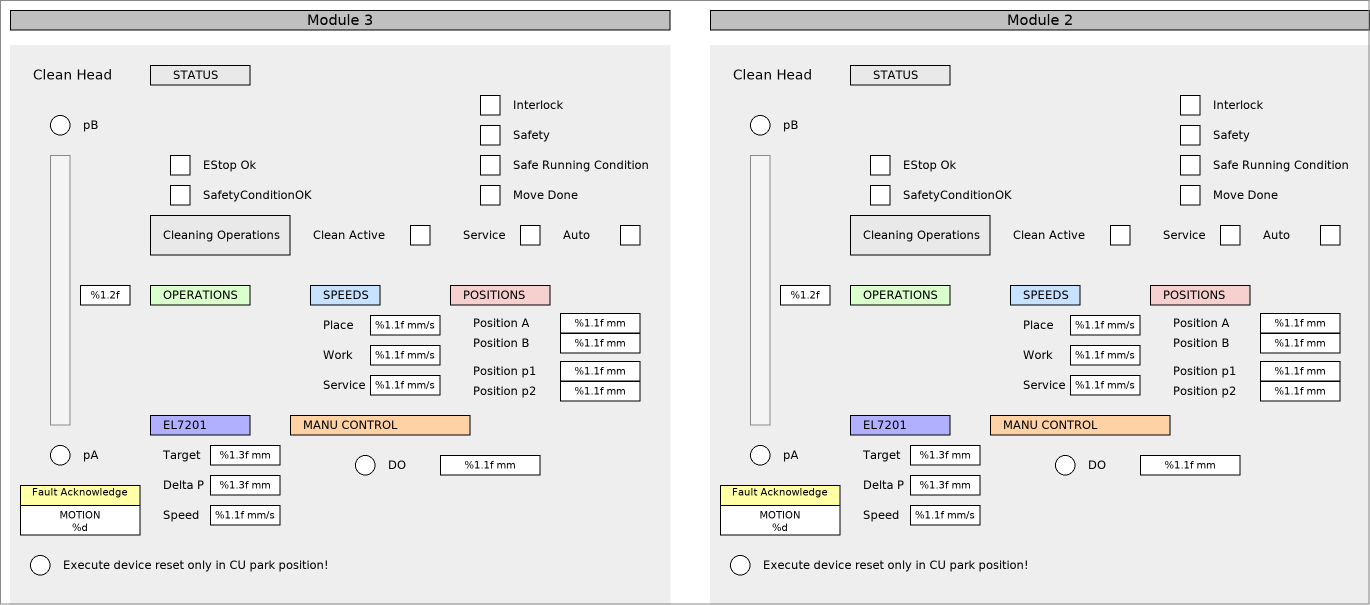
VISUALIZATION VISU_CLEAN_CH  // 1370x605
    Frame (10,45 660x560)
        shows _VISU_CLEAN_CH(m_Inst := 2)
    Rectangle (10,10 660x20), "Module 3"
    Rectangle (710,10 660x20), "Module 2"
    Frame (710,45 660x560)
        shows _VISU_CLEAN_CH(m_Inst := 1)
END_VISUALIZATION

// ---- VISUs/Projects/Machine/VISU_CLEAN_CU.TcVIS
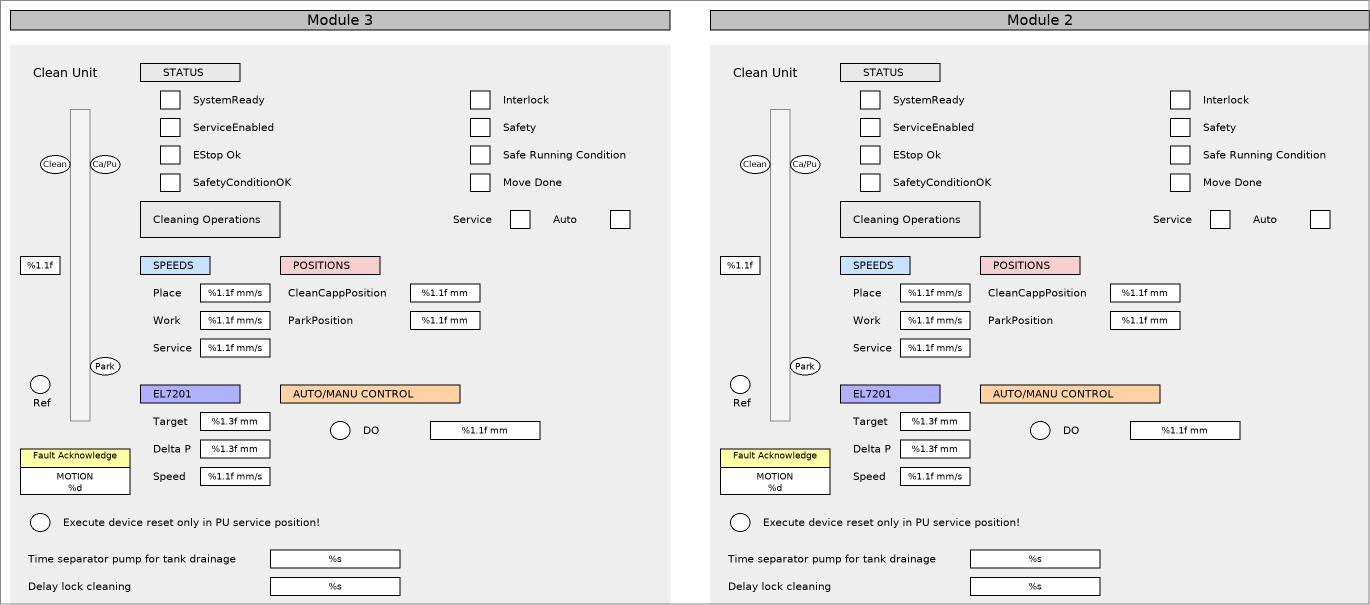
VISUALIZATION VISU_CLEAN_CU  // 1370x605
    Frame (10,45 660x560)
        shows _VISU_CLEAN_CU(m_Inst := 2)
    Rectangle (10,10 660x20), "Module 3"
    Rectangle (710,10 660x20), "Module 2"
    Frame (710,45 660x560)
        shows _VISU_CLEAN_CU(m_Inst := 1)
END_VISUALIZATION

// ---- VISUs/Projects/Machine/VISU_CLEAN_SEQUENCE.TcVIS
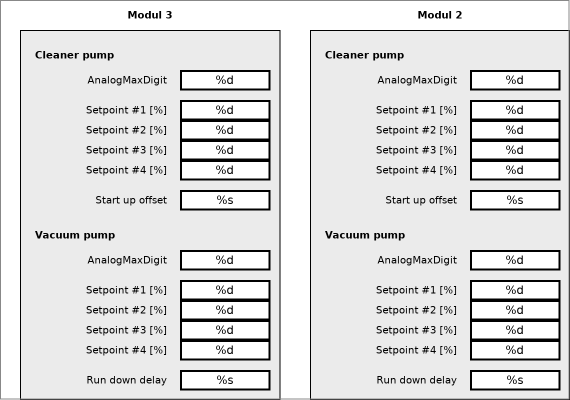
VISUALIZATION VISU_CLEAN_SEQUENCE  // 570x400
    Rectangle (20,30 260x370)
    Rectangle (180,70 90x20), "%d", text variable: PRG_MACHINE.fb_CleaningValvePump[2].lR_AnalogMaxDigitCleanerPump
        OnMouseDown: write the text variable via Default
    Rectangle (30,70 140x20), "AnalogMaxDigit"
    Rectangle (32,45 131x20), "Cleaner pump"
    Rectangle (180,100 90x20), "%d", text variable: PRG_MACHINE.fb_CleaningValvePump[2].lR_SetPoint1CleanerPump
        OnMouseDown: write the text variable via Default, min 0, max 100
    Rectangle (30,100 140x20), "Setpoint #1 [%]"
    Rectangle (180,120 90x20), "%d", text variable: PRG_MACHINE.fb_CleaningValvePump[2].lR_SetPoint2CleanerPump
        OnMouseDown: write the text variable via Default, min 0, max 100
    Rectangle (30,120 140x20), "Setpoint #2 [%]"
    Rectangle (180,140 90x20), "%d", text variable: PRG_MACHINE.fb_CleaningValvePump[2].lR_SetPoint3CleanerPump
        OnMouseDown: write the text variable via Default, min 0, max 100
    Rectangle (30,140 140x20), "Setpoint #3 [%]"
    Rectangle (180,160 90x20), "%d", text variable: PRG_MACHINE.fb_CleaningValvePump[2].lR_SetPoint4CleanerPump
        OnMouseDown: write the text variable via Default, min 0, max 100
    Rectangle (30,160 140x20), "Setpoint #4 [%]"
    Rectangle (180,250 90x20), "%d", text variable: PRG_MACHINE.fb_CleaningValvePump[2].lR_AnalogMaxDigitVacuumPump
        OnMouseDown: write the text variable via Default
    Rectangle (30,250 140x20), "AnalogMaxDigit"
    Rectangle (32,225 131x20), "Vacuum pump"
    Rectangle (180,280 90x20), "%d", text variable: PRG_MACHINE.fb_CleaningValvePump[2].lR_SetPoint1VacuumPump
        OnMouseDown: write the text variable via Default, min 0, max 100
    Rectangle (30,280 140x20), "Setpoint #1 [%]"
    Rectangle (180,300 90x20), "%d", text variable: PRG_MACHINE.fb_CleaningValvePump[2].lR_SetPoint2VacuumPump
        OnMouseDown: write the text variable via Default, min 0, max 100
    Rectangle (30,300 140x20), "Setpoint #2 [%]"
    Rectangle (180,320 90x20), "%d", text variable: PRG_MACHINE.fb_CleaningValvePump[2].lR_SetPoint3VacuumPump
        OnMouseDown: write the text variable via Default, min 0, max 100
    Rectangle (30,320 140x20), "Setpoint #3 [%]"
    Rectangle (180,340 90x20), "%d", text variable: PRG_MACHINE.fb_CleaningValvePump[2].lR_SetPoint4VacuumPump
        OnMouseDown: write the text variable via Default, min 0, max 100
    Rectangle (30,340 140x20), "Setpoint #4 [%]"
    Rectangle (180,190 90x20), "%s", text variable: PRG_MACHINE.fb_CleaningValvePump[2].tR_CleanerPumpOffset
        OnMouseDown: write the text variable via Default
    Rectangle (30,190 140x20), "Start up offset"
    Rectangle (180,370 90x20), "%s", text variable: PRG_MACHINE.fb_CleaningValvePump[2].tR_VacuumPumpDelay
        OnMouseDown: write the text variable via Default
    Rectangle (30,370 140x20), "Run down delay"
    Rectangle (310,30 260x370)
    Rectangle (470,70 90x20), "%d", text variable: PRG_MACHINE.fb_CleaningValvePump[1].lR_AnalogMaxDigitCleanerPump
        OnMouseDown: write the text variable via Default
    Rectangle (320,70 140x20), "AnalogMaxDigit"
    Rectangle (322,45 131x20), "Cleaner pump"
    Rectangle (470,100 90x20), "%d", text variable: PRG_MACHINE.fb_CleaningValvePump[1].lR_SetPoint1CleanerPump
        OnMouseDown: write the text variable via Default, min 0, max 100
    Rectangle (320,100 140x20), "Setpoint #1 [%]"
    Rectangle (470,120 90x20), "%d", text variable: PRG_MACHINE.fb_CleaningValvePump[1].lR_SetPoint2CleanerPump
        OnMouseDown: write the text variable via Default, min 0, max 100
    Rectangle (320,120 140x20), "Setpoint #2 [%]"
    Rectangle (470,140 90x20), "%d", text variable: PRG_MACHINE.fb_CleaningValvePump[1].lR_SetPoint3CleanerPump
        OnMouseDown: write the text variable via Default, min 0, max 100
    Rectangle (320,140 140x20), "Setpoint #3 [%]"
    Rectangle (470,160 90x20), "%d", text variable: PRG_MACHINE.fb_CleaningValvePump[1].lR_SetPoint4CleanerPump
        OnMouseDown: write the text variable via Default, min 0, max 100
    Rectangle (320,160 140x20), "Setpoint #4 [%]"
    Rectangle (470,250 90x20), "%d", text variable: PRG_MACHINE.fb_CleaningValvePump[1].lR_AnalogMaxDigitVacuumPump
        OnMouseDown: write the text variable via Default
    Rectangle (320,250 140x20), "AnalogMaxDigit"
    Rectangle (322,225 131x20), "Vacuum pump"
    Rectangle (470,280 90x20), "%d", text variable: PRG_MACHINE.fb_CleaningValvePump[1].lR_SetPoint1VacuumPump
        OnMouseDown: write the text variable via Default, min 0, max 100
    Rectangle (320,280 140x20), "Setpoint #1 [%]"
    Rectangle (470,300 90x20), "%d", text variable: PRG_MACHINE.fb_CleaningValvePump[1].lR_SetPoint2VacuumPump
        OnMouseDown: write the text variable via Default, min 0, max 100
    Rectangle (320,300 140x20), "Setpoint #2 [%]"
    Rectangle (470,320 90x20), "%d", text variable: PRG_MACHINE.fb_CleaningValvePump[1].lR_SetPoint3VacuumPump
        OnMouseDown: write the text variable via Default, min 0, max 100
    Rectangle (320,320 140x20), "Setpoint #3 [%]"
    Rectangle (470,340 90x20), "%d", text variable: PRG_MACHINE.fb_CleaningValvePump[1].lR_SetPoint4VacuumPump
        OnMouseDown: write the text variable via Default, min 0, max 100
    Rectangle (320,340 140x20), "Setpoint #4 [%]"
    Rectangle (470,190 90x20), "%s", text variable: PRG_MACHINE.fb_CleaningValvePump[1].tR_CleanerPumpOffset
        OnMouseDown: write the text variable via Default
    Rectangle (320,190 140x20), "Start up offset"
    Rectangle (470,370 90x20), "%s", text variable: PRG_MACHINE.fb_CleaningValvePump[1].tR_VacuumPumpDelay
        OnMouseDown: write the text variable via Default
    Rectangle (320,370 140x20), "Run down delay"
    Rectangle (310,5 260x20), "Modul 2"
    Rectangle (20,5 260x20), "Modul 3"
END_VISUALIZATION

// ---- VISUs/Projects/Machine/VISU_EXHAUST.TcVIS
